(* CoDeSys 2.3.9.31 project: tcWiesenrain23.pro *)
(* Libraries: C:\Users\root\Desktop\nww.wiesenrain23\lib\oscat_building_100.lib 12.1.13 01:09:34, C:\Users\root\Desktop\nww.wiesenrain23\lib\oscat_basic_333.lib 12.1.13 01:05:45, C:\Users\root\Desktop\nww.wiesenrain23\lib\ModbusRTU.lib 29.12.13 03:10:52, STANDARD.LIB 5.6.98 11:03:02, TcBase.lib 14.5.09 11:14:08, TcEtherCAT.lib 8.3.12 16:06:42, TcSUPS.lib 22.3.10 12:59:22, TcSystem.lib 27.2.12 14:08:36, TcUtilities.lib 10.1.13 19:12:12 *)

(* Task configuration *)
TASK Standard (PRIORITY := 1, INTERVAL := T#10ms);
	MAIN
END_TASK
TASK Slow (PRIORITY := 2, INTERVAL := T#200ms);
	MAIN_SLOW
END_TASK
TASK Fast (PRIORITY := 0, INTERVAL := T#1ms);
	MAIN_FAST
END_TASK

(* Global variable list: Global_Variables *)
VAR_GLOBAL
	A_TemperatureUnit: ARRAY [0..7] OF ST_TemperatureUnit := (
			id := KELVIN,   (* commonly used in scientific endeavors *)
			unit := 'Kelvin',
			symbol := 'K',
			f1 := 0,
			f2 := 273.16,
			offset := 0,
			scale := 1,
			inventor := 'William Thomson, 1st Baron Kelvin'
		), (
			id := GRAD_CELSIUS,   (* used by most of the world's population *)
			unit := 'Celsius',
			symbol := '°C',
			f1 := 0,
			f2 := 100,
			offset := 273.15,
			scale := 1,
			inventor := 'Anders Celsius'
		), (
			id := GRAD_FAHRENHEIT,   (* commonly used in the United States *)
			unit := 'Fahrenheit',
			symbol := '°F',
			f1 := 0,
			f2 := 96,
			offset := 255.3722222222222, (* 459.67 * 5 / 9 *)
			scale := 0.55555555555555555555,
			inventor := 'Daniel Gabriel Fahrenheit'
		), (
			id := GRAD_RANKINE,
			unit := 'Rankine',
			symbol := '°Ra',
			f1 := 0,
			f2 := 96,
			offset := 0,
			scale := 0.5555555555555555555,
			inventor := 'William John Macquorn Rankine'
		), (
			id := GRAD_DELISLE,
			unit := 'Delisle',
			symbol := '°De',
			f1 := 150,
			f2 := 0,
			offset := 373.15,
			scale := -0.66666666666666666666,
			inventor := 'Joseph-Nicolas Delisle'
		), (
			id := GRAD_REAUMUR,
			unit := 'Réaumur',
			symbol := '°Ré',
			f1 := 0,
			f2 := 80,
			offset := 273.15,
			scale := 1.25,
			inventor := 'René-Antoine Ferchault de Réaumur'
		), (
			id := GRAD_NEWTON,
			unit := 'Newton',
			symbol := '°N',
			f1 := 0,
			f2 := 33,
			offset := 273.15,
			scale := 0.66666666666666666666,
			inventor := 'Sir Isaac Newton'
		), (
			id := GRAD_ROMER,
			unit := 'Rømer',
			symbol := '°Rø',
			f1 := 0,
			f2 := 60,
			offset := 258.86428571428571428572, (* 273.15 - 7.5 * 40 / 21 *)
			scale := 1.90476190476190476190,
			inventor := 'Ole Christensen Rømer'
		);
END_VAR

(* Global variable list: Global_Variables_MODBUS *)
VAR_GLOBAL CONSTANT
	uiMaxCurrentDeviceSpace: UDINT := 99;
END_VAR

(* Global variable list: TwinCAT_Configuration *)
(* Generated automatically by TwinCAT - (read only) *)
VAR_CONFIG
	MAIN._bwmAussenW AT %IX296.0 : BOOL;
	MAIN._bwmAussenSO AT %IX296.1 : BOOL;
	MAIN._bwmEgGang AT %IX124.0 : BOOL;	(*  ~ {LinkedWith:TIID^KG-HV A1 X001 EtherCAT [rechts]^OG-UV A1 Ethercat->K-Bus [unten links] ^OG-UV A7^Kanal 9^EG-Gang BWM} *)
	MAIN._bwmEgWc AT %IX128.0 : BOOL;	(*  ~ {LinkedWith:TIID^KG-HV A1 X001 EtherCAT [rechts]^OG-UV A1 Ethercat->K-Bus [unten links] ^OG-UV A7^Kanal 11^EG-WC BWM} *)
	MAIN._bwmHobby AT %IX108.0 : BOOL;	(*  ~ {LinkedWith:TIID^KG-HV A1 X001 EtherCAT [rechts]^KG-HV A35 EtherCat->E-Bus [links]^KG-HV A? E-Bus->K-Bus^KG-HV A5^Kanal 1^Hobby BWM} *)
	MAIN._bwmKgGang AT %IX76.0 : BOOL;	(*  ~ {LinkedWith:TIID^KG-HV A1 K-Bus [rechts]^KG-HV A1 (K-Bus)^KG-HV A33^Kanal 2^KG-Gang BWM} *)
	MAIN._bwmKochen AT %IX206.0 : BOOL;	(*  ~ {LinkedWith:TIID^KG-HV A1 X001 EtherCAT [rechts]^OG-UV A1 Ethercat->K-Bus [unten links] ^OG-UV A7^Kanal 10^Kochen BWM} *)
	MAIN._bwmLager AT %IX108.1 : BOOL;	(*  ~ {LinkedWith:TIID^KG-HV A1 X001 EtherCAT [rechts]^KG-HV A35 EtherCat->E-Bus [links]^KG-HV A? E-Bus->K-Bus^KG-HV A5^Kanal 5^Lager BWM} *)
	MAIN._bwmOgGang AT %IX120.0 : BOOL;	(*  ~ {LinkedWith:TIID^KG-HV A1 X001 EtherCAT [rechts]^OG-UV A1 Ethercat->K-Bus [unten links] ^OG-UV A7^Kanal 16^OG-Gang BWM} *)
	MAIN._bwmWaschen AT %IX112.0 : BOOL;	(*  ~ {LinkedWith:TIID^KG-HV A1 X001 EtherCAT [rechts]^KG-HV A35 EtherCat->E-Bus [links]^KG-HV A? E-Bus->K-Bus^KG-HV A5^Kanal 2^Waschen BWM} *)
	MAIN._lichtEgGang_status AT %IB300 : USINT;	(*  ~ {LinkedWith:TIID^KG-HV A1 X001 EtherCAT [rechts]^OG-UV A? Ethercat->K-Bus [mitte rechts]^OG-UV A9a^Kanal 2^EgGang Licht Status} *)
	MAIN._lichtEgGang_dataIn AT %IB301 : INT;	(*  ~ {LinkedWith:TIID^KG-HV A1 X001 EtherCAT [rechts]^OG-UV A? Ethercat->K-Bus [mitte rechts]^OG-UV A9a^Kanal 2^EgGang Licht DataIn} *)
	MAIN._lichtEgWc_status AT %IB303 : USINT;	(*  ~ {LinkedWith:TIID^KG-HV A1 X001 EtherCAT [rechts]^OG-UV A? Ethercat->K-Bus [mitte rechts]^OG-UV A9b^Kanal 2^EgWc Licht Status} *)
	MAIN._lichtEgWc_dataIn AT %IB304 : INT;	(*  ~ {LinkedWith:TIID^KG-HV A1 X001 EtherCAT [rechts]^OG-UV A? Ethercat->K-Bus [mitte rechts]^OG-UV A9b^Kanal 2^EgWc Licht Daten Ein} *)
	MAIN._lichtHobby_status AT %IB306 : USINT;
	MAIN._lichtHobby_dataIn AT %IB307 : INT;
	MAIN._lichtKochen_status AT %IB309 : USINT;
	MAIN._lichtKochen_dataIn AT %IB310 : INT;
	MAIN._lichtLager_status AT %IB312 : USINT;
	MAIN._lichtLager_dataIn AT %IB313 : INT;
	MAIN._lichtOgGang_status AT %IB315 : USINT;
	MAIN._lichtOgGang_dataIn AT %IB316 : INT;
	MAIN._lichtWaschen_status AT %IB318 : USINT;	(*  ~ {LinkedWith:TIID^KG-HV A1 X001 EtherCAT [rechts]^KG-HV A35 EtherCat->E-Bus [links]^KG-HV A? E-Bus->K-Bus^KG-HV A8b^Kanal 2^Waschen Licht Status} *)
	MAIN._lichtWaschen_dataIn AT %IB319 : INT;	(*  ~ {LinkedWith:TIID^KG-HV A1 X001 EtherCAT [rechts]^KG-HV A35 EtherCat->E-Bus [links]^KG-HV A? E-Bus->K-Bus^KG-HV A8b^Kanal 2^Waschen Licht Daten Ein} *)
	MAIN._temperaturArbeiten_status AT %IB324 : USINT;	(*  ~ {LinkedWith:TIID^KG-HV A1 X001 EtherCAT [rechts]^OG-UV A? Ethercat->K-Bus [mitte rechts]^OG-UV A74a^Kanal 2^Arbeiten Temperatur Status} *)
	MAIN._temperaturArbeiten_dataIn AT %IB325 : INT;	(*  ~ {LinkedWith:TIID^KG-HV A1 X001 EtherCAT [rechts]^OG-UV A? Ethercat->K-Bus [mitte rechts]^OG-UV A74a^Kanal 2^Arbeiten Temperatur Daten Ein} *)
	MAIN._temperaturEgBad_status AT %IB327 : USINT;
	MAIN._temperaturEgBad_dataIn AT %IB328 : INT;
	MAIN._temperaturEgGangSM_status AT %IB330 : USINT;	(*  ~ {LinkedWith:TIID^KG-HV A1 X001 EtherCAT [rechts]^OG-UV A? Ethercat->K-Bus [mitte rechts]^OG-UV A9a^Kanal 1^EgGang TemperaturSM Status} *)
	MAIN._temperaturEgGangSM_dataIn AT %IB331 : INT;	(*  ~ {LinkedWith:TIID^KG-HV A1 X001 EtherCAT [rechts]^OG-UV A? Ethercat->K-Bus [mitte rechts]^OG-UV A9a^Kanal 1^EgGang TemperaturSM DataIn} *)
	MAIN._temperaturEgGangSO_status AT %IB333 : USINT;
	MAIN._temperaturEgGangSO_dataIn AT %IB334 : INT;
	MAIN._temperaturEgWc_status AT %IB336 : USINT;	(*  ~ {LinkedWith:TIID^KG-HV A1 X001 EtherCAT [rechts]^OG-UV A? Ethercat->K-Bus [mitte rechts]^OG-UV A9b^Kanal 1^EgWc Temperatur Status} *)
	MAIN._temperaturEgWc_dataIn AT %IB337 : INT;	(*  ~ {LinkedWith:TIID^KG-HV A1 X001 EtherCAT [rechts]^OG-UV A? Ethercat->K-Bus [mitte rechts]^OG-UV A9b^Kanal 1^EgWc Temperatur Daten Ein} *)
	MAIN._temperaturEssen_status AT %IB339 : USINT;
	MAIN._temperaturEssen_dataIn AT %IB340 : INT;
	MAIN._temperaturGaeste_status AT %IB342 : USINT;
	MAIN._temperaturGaeste_dataIn AT %IB343 : INT;
	MAIN._temperaturHobby_status AT %IB345 : USINT;
	MAIN._temperaturHobby_dataIn AT %IB346 : INT;
	MAIN._temperaturKochen_status AT %IB348 : USINT;
	MAIN._temperaturKochen_dataIn AT %IB349 : INT;
	MAIN._temperaturLager_status AT %IB351 : USINT;
	MAIN._temperaturLager_dataIn AT %IB352 : INT;
	MAIN._temperaturOgBad_status AT %IB354 : USINT;
	MAIN._temperaturOgBad_dataIn AT %IB355 : INT;
	MAIN._temperaturOgGang_status AT %IB357 : USINT;	(*  ~ {LinkedWith:TIID^KG-HV A1 X001 EtherCAT [rechts]^OG-UV A? Ethercat->K-Bus [mitte rechts]^OG-UV A73a^Kanal 1^OgGang Temperatur Status} *)
	MAIN._temperaturOgGang_dataIn AT %IB358 : INT;	(*  ~ {LinkedWith:TIID^KG-HV A1 X001 EtherCAT [rechts]^OG-UV A? Ethercat->K-Bus [mitte rechts]^OG-UV A73a^Kanal 1^OgGang Temperatur Daten Ein} *)
	MAIN._temperaturOgKind_status AT %IB360 : USINT;
	MAIN._temperaturOgKind_dataIn AT %IB361 : INT;
	MAIN._temperaturOgWc_status AT %IB363 : USINT;
	MAIN._temperaturOgWc_dataIn AT %IB364 : INT;
	MAIN._temperaturSchlafen_status AT %IB366 : USINT;	(*  ~ {LinkedWith:TIID^KG-HV A1 X001 EtherCAT [rechts]^OG-UV A? Ethercat->K-Bus [mitte rechts]^OG-UV A10a^Kanal 1^Schlafen Temperatur Status} *)
	MAIN._temperaturSchlafen_dataIn AT %IB367 : INT;	(*  ~ {LinkedWith:TIID^KG-HV A1 X001 EtherCAT [rechts]^OG-UV A? Ethercat->K-Bus [mitte rechts]^OG-UV A10a^Kanal 1^Schlafen Temperatur DataIn} *)
	MAIN._temperaturVorrat_status AT %IB369 : USINT;
	MAIN._temperaturVorrat_dataIn AT %IB370 : INT;
	MAIN._temperaturWaschenON_status AT %IB372 : USINT;	(*  ~ {LinkedWith:TIID^KG-HV A1 X001 EtherCAT [rechts]^KG-HV A35 EtherCat->E-Bus [links]^KG-HV A? E-Bus->K-Bus^KG-HV A8b^Kanal 1^WaschenO TemperaturN Status} *)
	MAIN._temperaturWaschenON_dataIn AT %IB373 : INT;	(*  ~ {LinkedWith:TIID^KG-HV A1 X001 EtherCAT [rechts]^KG-HV A35 EtherCat->E-Bus [links]^KG-HV A? E-Bus->K-Bus^KG-HV A8b^Kanal 1^WaschenO TemperaturN Daten Ein} *)
	MAIN._temperaturWaschenOS_status AT %IB375 : USINT;
	MAIN._temperaturWaschenOS_dataIn AT %IB376 : INT;
	MAIN._temperaturWohnen_status AT %IB378 : USINT;	(*  ~ {LinkedWith:TIID^KG-HV A1 X001 EtherCAT [rechts]^OG-UV A? Ethercat->K-Bus [mitte rechts]^OG-UV A10a^Kanal 2^Wohnen Temperatur Status} *)
	MAIN._temperaturWohnen_dataIn AT %IB379 : INT;	(*  ~ {LinkedWith:TIID^KG-HV A1 X001 EtherCAT [rechts]^OG-UV A? Ethercat->K-Bus [mitte rechts]^OG-UV A10a^Kanal 2^Wohnen Temperatur DataIn} *)
	MAIN._tasterArbeitenOO AT %IX206.1 : BOOL;	(*  ~ {LinkedWith:TIID^KG-HV A1 X001 EtherCAT [rechts]^OG-UV A1 Ethercat->K-Bus [unten links] ^OG-UV A6^Kanal 3^ArbeitenO TasterO} *)
	MAIN._tasterArbeitenOL AT %IX206.2 : BOOL;	(*  ~ {LinkedWith:TIID^KG-HV A1 X001 EtherCAT [rechts]^OG-UV A1 Ethercat->K-Bus [unten links] ^OG-UV A6^Kanal 4^ArbeitenO TasterL} *)
	MAIN._tasterArbeitenOR AT %IX206.3 : BOOL;	(*  ~ {LinkedWith:TIID^KG-HV A1 X001 EtherCAT [rechts]^OG-UV A1 Ethercat->K-Bus [unten links] ^OG-UV A6^Kanal 5^ArbeitenO TasterR} *)
	MAIN._tasterArbeitenSL AT %IX206.4 : BOOL;	(*  ~ {LinkedWith:TIID^KG-HV A1 X001 EtherCAT [rechts]^OG-UV A1 Ethercat->K-Bus [unten links] ^OG-UV A5^Kanal 11^ArbeitenS TasterL} *)
	MAIN._tasterArbeitenSR AT %IX206.5 : BOOL;	(*  ~ {LinkedWith:TIID^KG-HV A1 X001 EtherCAT [rechts]^OG-UV A1 Ethercat->K-Bus [unten links] ^OG-UV A5^Kanal 12^ArbeitenS TasterR} *)
	MAIN._tasterDgKind AT %IX206.6 : BOOL;
	MAIN._tasterEgBadL AT %IX132.1 : BOOL;	(*  ~ {LinkedWith:TIID^KG-HV A1 X001 EtherCAT [rechts]^OG-UV A1 Ethercat->K-Bus [unten links] ^OG-UV A5^Kanal 7^EG-Bad TasterL} *)
	MAIN._tasterEgBadR AT %IX132.0 : BOOL;	(*  ~ {LinkedWith:TIID^KG-HV A1 X001 EtherCAT [rechts]^OG-UV A1 Ethercat->K-Bus [unten links] ^OG-UV A5^Kanal 8^EG-Bad TasterR} *)
	MAIN._tasterEgGang AT %IX80.0 : BOOL;	(*  ~ {LinkedWith:TIID^KG-HV A1 K-Bus [rechts]^KG-HV A1 (K-Bus)^KG-HV A4^Kanal 10^EG-Gang Taster} *)
	MAIN._tasterEgWc AT %IX128.1 : BOOL;	(*  ~ {LinkedWith:TIID^KG-HV A1 X001 EtherCAT [rechts]^OG-UV A1 Ethercat->K-Bus [unten links] ^OG-UV A5^Kanal 6^EG-WC Taster} *)
	MAIN._tasterEssenO AT %IX140.0 : BOOL;	(*  ~ {LinkedWith:TIID^KG-HV A1 X001 EtherCAT [rechts]^OG-UV A1 Ethercat->K-Bus [unten links] ^OG-UV A4^Kanal 6^EssenS TasterO} *)
	MAIN._tasterEssenL AT %IX140.1 : BOOL;	(*  ~ {LinkedWith:TIID^KG-HV A1 X001 EtherCAT [rechts]^OG-UV A1 Ethercat->K-Bus [unten links] ^OG-UV A4^Kanal 7^EssenS TasterL} *)
	MAIN._tasterEssenR AT %IX140.2 : BOOL;	(*  ~ {LinkedWith:TIID^KG-HV A1 X001 EtherCAT [rechts]^OG-UV A1 Ethercat->K-Bus [unten links] ^OG-UV A4^Kanal 8^EssenS TasterR} *)
	MAIN._tasterGaesteO AT %IX136.0 : BOOL;	(*  ~ {LinkedWith:TIID^KG-HV A1 K-Bus [rechts]^KG-HV A1 (K-Bus)^OG-UV A72^Kanal 1^GaesteN TasterO} *)
	MAIN._tasterGaesteL AT %IX136.1 : BOOL;	(*  ~ {LinkedWith:TIID^KG-HV A1 K-Bus [rechts]^KG-HV A1 (K-Bus)^OG-UV A72^Kanal 2^GaesteN TasterL} *)
	MAIN._tasterGaesteR AT %IX136.2 : BOOL;	(*  ~ {LinkedWith:TIID^KG-HV A1 K-Bus [rechts]^KG-HV A1 (K-Bus)^OG-UV A72^Kanal 3^GaesteN TasterR} *)
	MAIN._tasterHeizen AT %IX76.1 : BOOL;	(*  ~ {LinkedWith:TIID^KG-HV A1 K-Bus [rechts]^KG-HV A1 (K-Bus)^KG-HV A4^Kanal 7^Heizen Taster} *)
	MAIN._tasterHobbyL AT %IX76.2 : BOOL;	(*  ~ {LinkedWith:TIID^KG-HV A1 K-Bus [rechts]^KG-HV A1 (K-Bus)^KG-HV A4^Kanal 5^Hobby TasterL} *)
	MAIN._tasterHobbyR AT %IX76.3 : BOOL;	(*  ~ {LinkedWith:TIID^KG-HV A1 K-Bus [rechts]^KG-HV A1 (K-Bus)^KG-HV A4^Kanal 6^Hobby TasterR} *)
	MAIN._tasterKochenOL AT %IX144.0 : BOOL;	(*  ~ {LinkedWith:TIID^KG-HV A1 X001 EtherCAT [rechts]^OG-UV A1 Ethercat->K-Bus [unten links] ^OG-UV A4^Kanal 4^KochenO TasterL} *)
	MAIN._tasterKochenOR AT %IX144.1 : BOOL;	(*  ~ {LinkedWith:TIID^KG-HV A1 X001 EtherCAT [rechts]^OG-UV A1 Ethercat->K-Bus [unten links] ^OG-UV A4^Kanal 5^KochenO TasterR} *)
	MAIN._tasterKochenWO AT %IX144.2 : BOOL;	(*  ~ {LinkedWith:TIID^KG-HV A1 X001 EtherCAT [rechts]^OG-UV A1 Ethercat->K-Bus [unten links] ^OG-UV A4^Kanal 1^KochenW TasterO} *)
	MAIN._tasterKochenWL AT %IX144.3 : BOOL;	(*  ~ {LinkedWith:TIID^KG-HV A1 X001 EtherCAT [rechts]^OG-UV A1 Ethercat->K-Bus [unten links] ^OG-UV A4^Kanal 2^KochenW TasterL} *)
	MAIN._tasterKochenWR AT %IX144.4 : BOOL;	(*  ~ {LinkedWith:TIID^KG-HV A1 X001 EtherCAT [rechts]^OG-UV A1 Ethercat->K-Bus [unten links] ^OG-UV A4^Kanal 3^KochenW TasterR} *)
	MAIN._tasterLagerNO AT %IX76.6 : BOOL;	(*  ~ {LinkedWith:TIID^KG-HV A1 K-Bus [rechts]^KG-HV A1 (K-Bus)^KG-HV A4^Kanal 9^LagerNO Taster} *)
	MAIN._tasterLagerS AT %IX76.7 : BOOL;	(*  ~ {LinkedWith:TIID^KG-HV A1 K-Bus [rechts]^KG-HV A1 (K-Bus)^KG-HV A4^Kanal 8^LagerS Taster} *)
	MAIN._tasterOgBadL AT %IX206.7 : BOOL;
	MAIN._tasterOgBadR AT %IX207.0 : BOOL;
	MAIN._tasterOgKindNO AT %IX207.1 : BOOL;
	MAIN._tasterOgKindNL AT %IX207.2 : BOOL;
	MAIN._tasterOgKindNR AT %IX207.3 : BOOL;
	MAIN._tasterOgKindWL AT %IX207.4 : BOOL;	(*  ~ {LinkedWith:TIID^KG-HV A1 X001 EtherCAT [rechts]^OG-UV A1 Ethercat->K-Bus [unten links] ^OG-UV A5^Kanal 9^OG-KindW TasterL} *)
	MAIN._tasterOgKindWR AT %IX207.5 : BOOL;	(*  ~ {LinkedWith:TIID^KG-HV A1 X001 EtherCAT [rechts]^OG-UV A1 Ethercat->K-Bus [unten links] ^OG-UV A5^Kanal 10^OG-KindW TasteR} *)
	MAIN._tasterOgWc AT %IX207.6 : BOOL;
	MAIN._tasterSchlafenOo AT %IX408.0 : BOOL;	(*  ~ {LinkedWith:TIID^KG-HV A1 X001 EtherCAT [rechts]^OG-UV A1 Ethercat->K-Bus [unten links] ^OG-UV A4^Kanal 12^SchlafenO TasterO} *)
	MAIN._tasterSchlafenOl AT %IX408.1 : BOOL;	(*  ~ {LinkedWith:TIID^KG-HV A1 X001 EtherCAT [rechts]^OG-UV A1 Ethercat->K-Bus [unten links] ^OG-UV A4^Kanal 13^SchlafenO TasterL} *)
	MAIN._tasterSchlafenOr AT %IX408.2 : BOOL;	(*  ~ {LinkedWith:TIID^KG-HV A1 X001 EtherCAT [rechts]^OG-UV A1 Ethercat->K-Bus [unten links] ^OG-UV A4^Kanal 14^SchlafenO TasterR} *)
	MAIN._tasterSchlafenWML AT %IX116.3 : BOOL;	(*  ~ {LinkedWith:TIID^KG-HV A1 X001 EtherCAT [rechts]^OG-UV A1 Ethercat->K-Bus [unten links] ^OG-UV A4^Kanal 15^SchlafenWM TasterL} *)
	MAIN._tasterSchlafenWMR AT %IX116.4 : BOOL;	(*  ~ {LinkedWith:TIID^KG-HV A1 X001 EtherCAT [rechts]^OG-UV A1 Ethercat->K-Bus [unten links] ^OG-UV A4^Kanal 16^SchlafenWM TasterR} *)
	MAIN._tasterSchlafenWNL AT %IX116.5 : BOOL;	(*  ~ {LinkedWith:TIID^KG-HV A1 X001 EtherCAT [rechts]^OG-UV A1 Ethercat->K-Bus [unten links] ^OG-UV A5^Kanal 1^SchlafenWN TasterL} *)
	MAIN._tasterSchlafenWNR AT %IX116.6 : BOOL;	(*  ~ {LinkedWith:TIID^KG-HV A1 X001 EtherCAT [rechts]^OG-UV A1 Ethercat->K-Bus [unten links] ^OG-UV A5^Kanal 2^SchlafenWN TasterR} *)
	MAIN._tasterSpeis AT %IX207.7 : BOOL;	(*  ~ {LinkedWith:TIID^KG-HV A1 X001 EtherCAT [rechts]^OG-UV A1 Ethercat->K-Bus [unten links] ^OG-UV A5^Kanal 16^Speis Tuerkontakt} *)
	MAIN._tasterWaschenL AT %IX76.4 : BOOL;	(*  ~ {LinkedWith:TIID^KG-HV A1 K-Bus [rechts]^KG-HV A1 (K-Bus)^KG-HV A4^Kanal 3^Waschen TasterL} *)
	MAIN._tasterWaschenR AT %IX76.5 : BOOL;	(*  ~ {LinkedWith:TIID^KG-HV A1 K-Bus [rechts]^KG-HV A1 (K-Bus)^KG-HV A4^Kanal 4^Waschen TasterR} *)
	MAIN._tasterWohnenOO AT %IX124.1 : BOOL;	(*  ~ {LinkedWith:TIID^KG-HV A1 X001 EtherCAT [rechts]^OG-UV A1 Ethercat->K-Bus [unten links] ^OG-UV A4^Kanal 9^WohnenO TasterO} *)
	MAIN._tasterWohnenOL AT %IX124.2 : BOOL;	(*  ~ {LinkedWith:TIID^KG-HV A1 X001 EtherCAT [rechts]^OG-UV A1 Ethercat->K-Bus [unten links] ^OG-UV A4^Kanal 10^WohnenO TasterL} *)
	MAIN._tasterWohnenOR AT %IX124.3 : BOOL;	(*  ~ {LinkedWith:TIID^KG-HV A1 X001 EtherCAT [rechts]^OG-UV A1 Ethercat->K-Bus [unten links] ^OG-UV A4^Kanal 11^WohnenO TasterR} *)
	MAIN._tasterWohnenWO AT %IX124.4 : BOOL;	(*  ~ {LinkedWith:TIID^KG-HV A1 X001 EtherCAT [rechts]^OG-UV A1 Ethercat->K-Bus [unten links] ^OG-UV A5^Kanal 3^WohnenW TasterO} *)
	MAIN._tasterWohnenWL AT %IX124.5 : BOOL;	(*  ~ {LinkedWith:TIID^KG-HV A1 X001 EtherCAT [rechts]^OG-UV A1 Ethercat->K-Bus [unten links] ^OG-UV A5^Kanal 4^WohnenW TasterL} *)
	MAIN._tasterWohnenWR AT %IX124.6 : BOOL;	(*  ~ {LinkedWith:TIID^KG-HV A1 X001 EtherCAT [rechts]^OG-UV A1 Ethercat->K-Bus [unten links] ^OG-UV A5^Kanal 5^WohnenW TasterR} *)
	MAIN._dimmerWohnenN_intensity AT %IB208 : REAL;
	MAIN._dimmerWohnenN_status AT %IB212 : USINT;	(*  ~ {LinkedWith:TIID^KG-HV A1 X001 EtherCAT [rechts]^OG-UV A? Ethercat->K-Bus [mitte rechts]^OG-UV A29^Kanal 1^WohnenM Lampe Status} *)
	MAIN._dimmerWohnenN_dataIn AT %IB213 : INT;	(*  ~ {LinkedWith:TIID^KG-HV A1 X001 EtherCAT [rechts]^OG-UV A? Ethercat->K-Bus [mitte rechts]^OG-UV A29^Kanal 1^WohnenM Lampe DataIn} *)
	MAIN._dimmerWohnenN_dataOut AT %QB24 : INT;	(*  ~ {LinkedWith:TIID^KG-HV A1 X001 EtherCAT [rechts]^OG-UV A? Ethercat->K-Bus [mitte rechts]^OG-UV A29^Kanal 1^WohnenM Lampe DataOut} *)
	MAIN._dimmerWohnenN_control AT %QB26 : USINT;	(*  ~ {LinkedWith:TIID^KG-HV A1 X001 EtherCAT [rechts]^OG-UV A? Ethercat->K-Bus [mitte rechts]^OG-UV A29^Kanal 1^WohnenM Lampe Control} *)
	MAIN._dimmerEgBadSM_intensity AT %IB216 : REAL;
	MAIN._dimmerEgBadSM_status AT %IB220 : USINT;	(*  ~ {LinkedWith:TIID^KG-HV A1 X001 EtherCAT [rechts]^OG-UV A? Ethercat->K-Bus [mitte rechts]^OG-UV A32^Kanal 1^EgBad LichtSM Status} *)
	MAIN._dimmerEgBadSM_dataIn AT %IB221 : INT;	(*  ~ {LinkedWith:TIID^KG-HV A1 X001 EtherCAT [rechts]^OG-UV A? Ethercat->K-Bus [mitte rechts]^OG-UV A32^Kanal 1^EgBad LichtSM Daten Ein} *)
	MAIN._dimmerEgBadSM_dataOut AT %QB36 : INT;	(*  ~ {LinkedWith:TIID^KG-HV A1 X001 EtherCAT [rechts]^OG-UV A? Ethercat->K-Bus [mitte rechts]^OG-UV A32^Kanal 1^EgBad LichtSM Daten Aus} *)
	MAIN._dimmerEgBadSM_control AT %QB38 : USINT;	(*  ~ {LinkedWith:TIID^KG-HV A1 X001 EtherCAT [rechts]^OG-UV A? Ethercat->K-Bus [mitte rechts]^OG-UV A32^Kanal 1^EgBad LichtSM Kontrolle} *)
	MAIN._lampeEgBadOM AT %QX20.1 : BOOL;	(*  ~ {LinkedWith:TIID^KG-HV A1 X001 EtherCAT [rechts]^OG-UV A1 Ethercat->K-Bus [unten links] ^OG-UV A31^Kanal 2^EG-BadOM Lampe} *)
	MAIN._lampeEgGang AT %QX20.2 : BOOL;	(*  ~ {LinkedWith:TIID^KG-HV A1 X001 EtherCAT [rechts]^OG-UV A1 Ethercat->K-Bus [unten links] ^OG-UV A24^Kanal 1^EG-Gang Lampen} *)
	MAIN._lampeEgWc AT %QX20.3 : BOOL;	(*  ~ {LinkedWith:TIID^KG-HV A1 X001 EtherCAT [rechts]^OG-UV A1 Ethercat->K-Bus [unten links] ^OG-UV A31^Kanal 1^EG-WC Lampe} *)
	MAIN._lampeEssenM AT %QX20.4 : BOOL;	(*  ~ {LinkedWith:TIID^KG-HV A1 X001 EtherCAT [rechts]^OG-UV A1 Ethercat->K-Bus [unten links] ^OG-UV A14^Kanal 1^EssenM Lampe} *)
	MAIN._lampeEssenS AT %QX20.5 : BOOL;	(*  ~ {LinkedWith:TIID^KG-HV A1 X001 EtherCAT [rechts]^OG-UV A1 Ethercat->K-Bus [unten links] ^OG-UV A14^Kanal 2^EssenS Lampe} *)
	MAIN._lampeKochenSW AT %QX32.0 : BOOL;	(*  ~ {LinkedWith:TIID^KG-HV A1 X001 EtherCAT [rechts]^OG-UV A1 Ethercat->K-Bus [unten links] ^OG-UV A24^Kanal 2^KochenSW Lampe} *)
	MAIN._lampeOgGang AT %QX20.6 : BOOL;	(*  ~ {LinkedWith:TIID^KG-HV A1 K-Bus [rechts]^KG-HV A1 (K-Bus)^OG-UV A40^Kanal 1^OG-Gang Lampe} *)
	MAIN._lampeEgOgStiege AT %QX52.0 : BOOL;	(*  ~ {LinkedWith:TIID^KG-HV A1 K-Bus [rechts]^KG-HV A1 (K-Bus)^OG-UV A40^Kanal 2^EG-OG-Stiege Lampe} *)
	MAIN._lampeSchlafenS AT %QX20.0 : BOOL;	(*  ~ {LinkedWith:TIID^KG-HV A1 X001 EtherCAT [rechts]^OG-UV A1 Ethercat->K-Bus [unten links] ^OG-UV A28^Kanal 1^SchlafenS Lampen} *)
	MAIN._lampeWohnenM AT %QX28.0 : BOOL;	(*  ~ {LinkedWith:TIID^KG-HV A1 X001 EtherCAT [rechts]^OG-UV A1 Ethercat->K-Bus [unten links] ^OG-UV A28^Kanal 2^WohnenM Lampe} *)
	MAIN.heizenHK1.mischer AT %QB12 : INT;
	MAIN.heizenHK1.pumpe AT %QB14 : INT;
	MAIN.heizenHK2.mischer AT %QB16 : INT;
	MAIN.heizenHK2.pumpe AT %QB18 : INT;
	MAIN.egBadJalousie.Qu AT %QX92.0 : BOOL;	(*  ~ {LinkedWith:TIID^KG-HV A1 K-Bus [rechts]^KG-HV A1 (K-Bus)^OG-UV A59^Kanal 1^EG-Bad JalousieAuf} *)
	MAIN.egBadJalousie.Qd AT %QX92.1 : BOOL;	(*  ~ {LinkedWith:TIID^KG-HV A1 K-Bus [rechts]^KG-HV A1 (K-Bus)^OG-UV A59^Kanal 2^EG-Bad JalousieAb} *)
	MAIN.essenJalousie.Qu AT %QX92.2 : BOOL;	(*  ~ {LinkedWith:TIID^KG-HV A1 X001 EtherCAT [rechts]^OG-UV A1 Ethercat->K-Bus [unten links] ^OG-UV A65^Kanal 1^Essen JalousieAuf} *)
	MAIN.essenJalousie.Qd AT %QX92.3 : BOOL;	(*  ~ {LinkedWith:TIID^KG-HV A1 X001 EtherCAT [rechts]^OG-UV A1 Ethercat->K-Bus [unten links] ^OG-UV A65^Kanal 2^Essen JalousieAb} *)
	MAIN.kochenJalousieS.Qu AT %QX92.4 : BOOL;	(*  ~ {LinkedWith:TIID^KG-HV A1 X001 EtherCAT [rechts]^OG-UV A1 Ethercat->K-Bus [unten links] ^OG-UV A66^Kanal 1^KochenS JalousieAuf} *)
	MAIN.kochenJalousieS.Qd AT %QX92.5 : BOOL;	(*  ~ {LinkedWith:TIID^KG-HV A1 X001 EtherCAT [rechts]^OG-UV A1 Ethercat->K-Bus [unten links] ^OG-UV A66^Kanal 2^KochenS JalousieAb} *)
	MAIN.kochenJalousieO.Qu AT %QX92.6 : BOOL;	(*  ~ {LinkedWith:TIID^KG-HV A1 X001 EtherCAT [rechts]^OG-UV A1 Ethercat->K-Bus [unten links] ^OG-UV A67^Kanal 1^KochenO JalousieAuf} *)
	MAIN.kochenJalousieO.Qd AT %QX92.7 : BOOL;	(*  ~ {LinkedWith:TIID^KG-HV A1 X001 EtherCAT [rechts]^OG-UV A1 Ethercat->K-Bus [unten links] ^OG-UV A67^Kanal 2^KochenO JalousieAb} *)
	MAIN.schlafenJalousieN.Qu AT %QX88.2 : BOOL;	(*  ~ {LinkedWith:TIID^KG-HV A1 K-Bus [rechts]^KG-HV A1 (K-Bus)^OG-UV A60^Kanal 1^SchlafenN JalousieAuf} *)
	MAIN.schlafenJalousieN.Qd AT %QX88.3 : BOOL;	(*  ~ {LinkedWith:TIID^KG-HV A1 K-Bus [rechts]^KG-HV A1 (K-Bus)^OG-UV A60^Kanal 2^SchlafenN JalousieAb} *)
	MAIN.schlafenJalousieW.Qu AT %QX88.4 : BOOL;	(*  ~ {LinkedWith:TIID^KG-HV A1 K-Bus [rechts]^KG-HV A1 (K-Bus)^OG-UV A61^Kanal 1^SchlafenW JalousieAuf} *)
	MAIN.schlafenJalousieW.Qd AT %QX88.5 : BOOL;	(*  ~ {LinkedWith:TIID^KG-HV A1 K-Bus [rechts]^KG-HV A1 (K-Bus)^OG-UV A61^Kanal 2^SchlafenW JalousieAb} *)
	MAIN.wohnenJalousieS.Qu AT %QX93.0 : BOOL;	(*  ~ {LinkedWith:TIID^KG-HV A1 X001 EtherCAT [rechts]^OG-UV A1 Ethercat->K-Bus [unten links] ^OG-UV A64^Kanal 1^WohnenS JalousieAuf} *)
	MAIN.wohnenJalousieS.Qd AT %QX93.1 : BOOL;	(*  ~ {LinkedWith:TIID^KG-HV A1 X001 EtherCAT [rechts]^OG-UV A1 Ethercat->K-Bus [unten links] ^OG-UV A64^Kanal 2^WohnenS JalousieAb} *)
	MAIN.wohnenJalousieWa.Qu AT %QX93.2 : BOOL;	(*  ~ {LinkedWith:TIID^KG-HV A1 K-Bus [rechts]^KG-HV A1 (K-Bus)^OG-UV A62^Kanal 1^WohnenWa JalousieAuf} *)
	MAIN.wohnenJalousieWa.Qd AT %QX93.3 : BOOL;	(*  ~ {LinkedWith:TIID^KG-HV A1 K-Bus [rechts]^KG-HV A1 (K-Bus)^OG-UV A62^Kanal 2^WohnenWa JalousieAb} *)
	MAIN.wohnenJalousieWb.Qu AT %QX93.4 : BOOL;	(*  ~ {LinkedWith:TIID^KG-HV A1 K-Bus [rechts]^KG-HV A1 (K-Bus)^OG-UV A63^Kanal 1^WohnenWb JalousieAuf} *)
	MAIN.wohnenJalousieWb.Qd AT %QX93.5 : BOOL;	(*  ~ {LinkedWith:TIID^KG-HV A1 K-Bus [rechts]^KG-HV A1 (K-Bus)^OG-UV A63^Kanal 2^WohnenWb JalousieAb} *)
	MAIN.arbeitenJalousieN.Qu AT %QX100.0 : BOOL;
	MAIN.arbeitenJalousieN.Qd AT %QX100.1 : BOOL;
	MAIN.arbeitenJalousieW.Qu AT %QX100.2 : BOOL;
	MAIN.arbeitenJalousieW.Qd AT %QX100.3 : BOOL;
	MAIN.arbeitenJalousieS.Qu AT %QX100.4 : BOOL;
	MAIN.arbeitenJalousieS.Qd AT %QX100.5 : BOOL;
	MAIN.gaesteJalousieO.Qu AT %QX100.6 : BOOL;
	MAIN.gaesteJalousieO.Qd AT %QX100.7 : BOOL;
	MAIN.gaesteJalousieS.Qu AT %QX101.0 : BOOL;
	MAIN.gaesteJalousieS.Qd AT %QX101.1 : BOOL;
	MAIN.ogBadJalousie.Qu AT %QX96.0 : BOOL;	(*  ~ {LinkedWith:TIID^KG-HV A1 K-Bus [rechts]^KG-HV A1 (K-Bus)^OG-UV A82^Kanal 1^OG-Bad JalousieAuf} *)
	MAIN.ogBadJalousie.Qd AT %QX96.1 : BOOL;	(*  ~ {LinkedWith:TIID^KG-HV A1 K-Bus [rechts]^KG-HV A1 (K-Bus)^OG-UV A82^Kanal 2^OG-Bad JalousieAb} *)
	MAIN.ogKindJalousieS.Qu AT %QX101.2 : BOOL;
	MAIN.ogKindJalousieS.Qd AT %QX101.3 : BOOL;
	MAIN.ogKindJalousieW.Qu AT %QX101.4 : BOOL;
	MAIN.ogKindJalousieW.Qd AT %QX101.5 : BOOL;
	MAIN_FAST.fbFroeling.modbusMaster.InData AT %IB384 : MB_KL6inData22B;
	MAIN_FAST.fbFroeling.modbusMaster.OutData AT %QB56 : MB_KL6outData22B;
	MAIN_FAST.uiStateCX5000 AT %IB224 : UINT;	(*  ~ {LinkedWith:TIID^KG-HV A1 K-Bus [rechts]^KG-HV A1 (K-Bus)^Eingänge^State} *)
	MAIN_FAST.uiControlCX5000 AT %QB40 : UINT;	(*  ~ {LinkedWith:TIID^KG-HV A1 K-Bus [rechts]^KG-HV A1 (K-Bus)^Ausgänge^Ctrl} *)
	MAIN_FAST.iVoltagePhase1 AT %IB226 : ARRAY [0..9] OF INT;	(*  ~ {LinkedWith:TIID^KG-HV A1 X001 EtherCAT [rechts]^KG-HV A35 EtherCat->E-Bus [links]^KG-HV A18^L1 Voltage Samples^U1 SAMPLES} *)
	MAIN_FAST.iVoltagePhase2 AT %IB246 : ARRAY [0..9] OF INT;	(*  ~ {LinkedWith:TIID^KG-HV A1 X001 EtherCAT [rechts]^KG-HV A35 EtherCat->E-Bus [links]^KG-HV A18^L2 Voltage Samples^U2 SAMPLES} *)
	MAIN_FAST.iVoltagePhase3 AT %IB266 : ARRAY [0..9] OF INT;	(*  ~ {LinkedWith:TIID^KG-HV A1 X001 EtherCAT [rechts]^KG-HV A35 EtherCat->E-Bus [links]^KG-HV A18^L3 Voltage Samples^U3 SAMPLES} *)
	MAIN_FAST.uliStartTimeNextLatch AT %IB286 : ARRAY [0..1] OF UDINT;	(*  ~ {LinkedWith:TIID^KG-HV A1 X001 EtherCAT [rechts]^KG-HV A35 EtherCat->E-Bus [links]^KG-HV A18^AI Timestamp NextSync1Time^StartTimeNextLatch} *)
	MAIN_FAST.bWcState AT %IX294.0 : BOOL;	(*  ~ {LinkedWith:TIID^KG-HV A1 X001 EtherCAT [rechts]^KG-HV A35 EtherCat->E-Bus [links]^KG-HV A18^WcState^WcState} *)
	MAIN_FAST.fbA28CH1.bRelay AT %QX42.0 : BOOL;	(*  ~ {LinkedWith:TIID^KG-HV A1 K-Bus [rechts]^KG-HV A1 (K-Bus)^KG-HV A28^Kanal 1^Heizen PumpeSolar} *)
	MAIN_FAST.fbA28CH2.bRelay AT %QX42.1 : BOOL;	(*  ~ {LinkedWith:TIID^KG-HV A1 K-Bus [rechts]^KG-HV A1 (K-Bus)^KG-HV A28^Kanal 2^Heizen PumpeWarmwasser} *)
	MAIN_FAST.fbA29CH1.bRelay AT %QX42.2 : BOOL;	(*  ~ {LinkedWith:TIID^KG-HV A1 K-Bus [rechts]^KG-HV A1 (K-Bus)^KG-HV A29^Kanal 1^Heizen PumpePufferladung} *)
	MAIN_FAST.fbA29CH2.bRelay AT %QX42.3 : BOOL;	(*  ~ {LinkedWith:TIID^KG-HV A1 K-Bus [rechts]^KG-HV A1 (K-Bus)^KG-HV A29^Kanal 2^Heizen PumpeHeizkreis2} *)
	MAIN_FAST.fbA30CH1.bRelay AT %QX42.4 : BOOL;	(*  ~ {LinkedWith:TIID^KG-HV A1 K-Bus [rechts]^KG-HV A1 (K-Bus)^KG-HV A30^Kanal 1^Heizen MischerPuffer} *)
	MAIN_FAST.fbA30CH2.bRelay AT %QX42.5 : BOOL;	(*  ~ {LinkedWith:TIID^KG-HV A1 K-Bus [rechts]^KG-HV A1 (K-Bus)^KG-HV A30^Kanal 2^Heizen MischerSolar} *)
	MAIN_FAST.fbA31CH1.bRelay AT %QX42.6 : BOOL;	(*  ~ {LinkedWith:TIID^KG-HV A1 K-Bus [rechts]^KG-HV A1 (K-Bus)^KG-HV A31 (reserve)^Kanal 1^Ausgang} *)
	MAIN_FAST.fbA31CH2.bRelay AT %QX42.7 : BOOL;	(*  ~ {LinkedWith:TIID^KG-HV A1 K-Bus [rechts]^KG-HV A1 (K-Bus)^KG-HV A31 (reserve)^Kanal 2^Ausgang} *)
	MAIN_FAST.fbA32CH1.bRelay AT %QX43.0 : BOOL;	(*  ~ {LinkedWith:TIID^KG-HV A1 K-Bus [rechts]^KG-HV A1 (K-Bus)^KG-HV A32^Kanal 1^Waschen Tauchpumpe} *)
	MAIN_FAST.fbA32CH2.bRelay AT %QX43.1 : BOOL;	(*  ~ {LinkedWith:TIID^KG-HV A1 K-Bus [rechts]^KG-HV A1 (K-Bus)^KG-HV A32^Kanal 2^Ausgang} *)
	MAIN_FAST.fbA20CH1.bRelay AT %QX43.2 : BOOL;	(*  ~ {LinkedWith:TIID^KG-HV A1 K-Bus [rechts]^KG-HV A1 (K-Bus)^KG-HV A20^Kanal 1^KG-Gang Lampe} *)
	MAIN_FAST.fbA20CH2.bRelay AT %QX43.3 : BOOL;	(*  ~ {LinkedWith:TIID^KG-HV A1 K-Bus [rechts]^KG-HV A1 (K-Bus)^KG-HV A20^Kanal 2^KG-EG-Stiege Lampe} *)
	MAIN_FAST.fbA21CH1.bRelay AT %QX43.4 : BOOL;	(*  ~ {LinkedWith:TIID^KG-HV A1 K-Bus [rechts]^KG-HV A1 (K-Bus)^KG-HV A21^Kanal 1^Lager Lampe} *)
	MAIN_FAST.fbA21CH2.bRelay AT %QX43.5 : BOOL;	(*  ~ {LinkedWith:TIID^KG-HV A1 K-Bus [rechts]^KG-HV A1 (K-Bus)^KG-HV A21^Kanal 2^Ausgang} *)
	MAIN_FAST.fbA23CH1.bRelay AT %QX43.6 : BOOL;	(*  ~ {LinkedWith:TIID^KG-HV A1 K-Bus [rechts]^KG-HV A1 (K-Bus)^KG-HV A23^Kanal 1^Heizen Lampe} *)
	MAIN_FAST.fbA23CH2.bRelay AT %QX43.7 : BOOL;	(*  ~ {LinkedWith:TIID^KG-HV A1 K-Bus [rechts]^KG-HV A1 (K-Bus)^KG-HV A23^Kanal 2^WaschenS Lampe} *)
	MAIN_FAST.fbA24CH1.bRelay AT %QX44.0 : BOOL;	(*  ~ {LinkedWith:TIID^KG-HV A1 K-Bus [rechts]^KG-HV A1 (K-Bus)^KG-HV A24^Kanal 1^WaschenN Lampe} *)
	MAIN_FAST.fbA24CH2.bRelay AT %QX44.1 : BOOL;	(*  ~ {LinkedWith:TIID^KG-HV A1 K-Bus [rechts]^KG-HV A1 (K-Bus)^KG-HV A24^Kanal 2^HobbyN Lampe} *)
	MAIN_FAST.fbA25CH1.bRelay AT %QX44.2 : BOOL;	(*  ~ {LinkedWith:TIID^KG-HV A1 K-Bus [rechts]^KG-HV A1 (K-Bus)^KG-HV A25^Kanal 1^Vorrat Lampe} *)
	MAIN_FAST.fbA25CH2.bRelay AT %QX44.3 : BOOL;	(*  ~ {LinkedWith:TIID^KG-HV A1 K-Bus [rechts]^KG-HV A1 (K-Bus)^KG-HV A25^Kanal 2^HobbyS Lampe} *)
	MAIN_FAST.fbA26CH1.bRelay AT %QX44.4 : BOOL;	(*  ~ {LinkedWith:TIID^KG-HV A1 K-Bus [rechts]^KG-HV A1 (K-Bus)^KG-HV A26^Kanal 1^Ausgang} *)
	MAIN_FAST.fbA26CH2.bRelay AT %QX44.5 : BOOL;	(*  ~ {LinkedWith:TIID^KG-HV A1 K-Bus [rechts]^KG-HV A1 (K-Bus)^KG-HV A26^Kanal 2^Ausgang} *)
	MAIN_FAST.fbA38OGCH1.bRelay AT %QX44.6 : BOOL;	(*  ~ {LinkedWith:TIID^KG-HV A1 K-Bus [rechts]^KG-HV A1 (K-Bus)^OG-UV A38^Kanal 1^Ausgang} *)
	MAIN_FAST.fbA38OGCH2.bRelay AT %QX44.7 : BOOL;	(*  ~ {LinkedWith:TIID^KG-HV A1 K-Bus [rechts]^KG-HV A1 (K-Bus)^OG-UV A38^Kanal 2^Ausgang} *)
	MAIN_FAST.fbA41OGCH1.bRelay AT %QX45.0 : BOOL;	(*  ~ {LinkedWith:TIID^KG-HV A1 K-Bus [rechts]^KG-HV A1 (K-Bus)^OG-UV A41^Kanal 1^OG-BadO Lampe} *)
	MAIN_FAST.fbA41OGCH2.bRelay AT %QX45.1 : BOOL;	(*  ~ {LinkedWith:TIID^KG-HV A1 K-Bus [rechts]^KG-HV A1 (K-Bus)^OG-UV A41^Kanal 2^Ausgang} *)
	MAIN_FAST.fbA43OGCH1.bRelay AT %QX45.2 : BOOL;	(*  ~ {LinkedWith:TIID^KG-HV A1 K-Bus [rechts]^KG-HV A1 (K-Bus)^OG-UV A43^Kanal 1^Ausgang} *)
	MAIN_FAST.fbA43OGCH2.bRelay AT %QX45.3 : BOOL;	(*  ~ {LinkedWith:TIID^KG-HV A1 K-Bus [rechts]^KG-HV A1 (K-Bus)^OG-UV A43^Kanal 2^Ausgang} *)
	MAIN_FAST.fbA44OGCH1.bRelay AT %QX45.4 : BOOL;	(*  ~ {LinkedWith:TIID^KG-HV A1 K-Bus [rechts]^KG-HV A1 (K-Bus)^OG-UV A44^Kanal 1^OG-KindN LampenWO} *)
	MAIN_FAST.fbA44OGCH2.bRelay AT %QX45.5 : BOOL;	(*  ~ {LinkedWith:TIID^KG-HV A1 K-Bus [rechts]^KG-HV A1 (K-Bus)^OG-UV A44^Kanal 2^OG-KindS LampenWO} *)
	MAIN_FAST.fbA45OGCH1.bRelay AT %QX45.6 : BOOL;	(*  ~ {LinkedWith:TIID^KG-HV A1 K-Bus [rechts]^KG-HV A1 (K-Bus)^OG-UV A45^Kanal 1^OG-KindN LampeM} *)
	MAIN_FAST.fbA45OGCH2.bRelay AT %QX45.7 : BOOL;	(*  ~ {LinkedWith:TIID^KG-HV A1 K-Bus [rechts]^KG-HV A1 (K-Bus)^OG-UV A45^Kanal 2^DG-KindO Lampe} *)
	MAIN_FAST.fbA48OGCH1.bRelay AT %QX46.0 : BOOL;	(*  ~ {LinkedWith:TIID^KG-HV A1 K-Bus [rechts]^KG-HV A1 (K-Bus)^OG-UV A48^Kanal 1^GaesteW LampenNS} *)
	MAIN_FAST.fbA48OGCH2.bRelay AT %QX46.1 : BOOL;	(*  ~ {LinkedWith:TIID^KG-HV A1 K-Bus [rechts]^KG-HV A1 (K-Bus)^OG-UV A48^Kanal 2^GaesteO LampenNS} *)
	MAIN_FAST.fbA49OGCH1.bRelay AT %QX46.2 : BOOL;	(*  ~ {LinkedWith:TIID^KG-HV A1 K-Bus [rechts]^KG-HV A1 (K-Bus)^OG-UV A49^Kanal 1^OG-BadDecke Lampen} *)
	MAIN_FAST.fbA49OGCH2.bRelay AT %QX46.3 : BOOL;	(*  ~ {LinkedWith:TIID^KG-HV A1 K-Bus [rechts]^KG-HV A1 (K-Bus)^OG-UV A49^Kanal 2^OG-BadON Lampe} *)
	MAIN_FAST.fbA50OGCH1.bRelay AT %QX46.4 : BOOL;	(*  ~ {LinkedWith:TIID^KG-HV A1 K-Bus [rechts]^KG-HV A1 (K-Bus)^OG-UV A50^Kanal 1^OG-WC Lampe} *)
	MAIN_FAST.fbA50OGCH2.bRelay AT %QX46.5 : BOOL;	(*  ~ {LinkedWith:TIID^KG-HV A1 K-Bus [rechts]^KG-HV A1 (K-Bus)^OG-UV A50^Kanal 2^Ausgang} *)
	MAIN_FAST.fbA52OGCH1.bRelay AT %QX46.6 : BOOL;	(*  ~ {LinkedWith:TIID^KG-HV A1 K-Bus [rechts]^KG-HV A1 (K-Bus)^OG-UV A52^Kanal 1^Ausgang} *)
	MAIN_FAST.fbA52OGCH2.bRelay AT %QX46.7 : BOOL;	(*  ~ {LinkedWith:TIID^KG-HV A1 K-Bus [rechts]^KG-HV A1 (K-Bus)^OG-UV A52^Kanal 2^Ausgang} *)
	MAIN_FAST.fbA53OGCH1.bRelay AT %QX47.0 : BOOL;	(*  ~ {LinkedWith:TIID^KG-HV A1 K-Bus [rechts]^KG-HV A1 (K-Bus)^OG-UV A53^Kanal 1^Balkon Steckdose} *)
	MAIN_FAST.fbA53OGCH2.bRelay AT %QX47.1 : BOOL;	(*  ~ {LinkedWith:TIID^KG-HV A1 K-Bus [rechts]^KG-HV A1 (K-Bus)^OG-UV A53^Kanal 2^Balkon Lampe} *)
	MAIN_FAST.fbA55OGCH1.bRelay AT %QX47.2 : BOOL;	(*  ~ {LinkedWith:TIID^KG-HV A1 K-Bus [rechts]^KG-HV A1 (K-Bus)^OG-UV A55^Kanal 1^AussenO Lampe} *)
	MAIN_FAST.fbA55OGCH2.bRelay AT %QX47.3 : BOOL;	(*  ~ {LinkedWith:TIID^KG-HV A1 K-Bus [rechts]^KG-HV A1 (K-Bus)^OG-UV A55^Kanal 2^AussenOS Lampe} *)
	MAIN_FAST.fbA56OGCH1.bRelay AT %QX47.4 : BOOL;	(*  ~ {LinkedWith:TIID^KG-HV A1 K-Bus [rechts]^KG-HV A1 (K-Bus)^OG-UV A56^Kanal 1^AussenWS Lampe} *)
	MAIN_FAST.fbA56OGCH2.bRelay AT %QX47.5 : BOOL;	(*  ~ {LinkedWith:TIID^KG-HV A1 K-Bus [rechts]^KG-HV A1 (K-Bus)^OG-UV A56^Kanal 2^AussenW Lampe} *)
	MAIN_FAST.fbA57OGCH1.bRelay AT %QX47.6 : BOOL;	(*  ~ {LinkedWith:TIID^KG-HV A1 K-Bus [rechts]^KG-HV A1 (K-Bus)^OG-UV A57^Kanal 1^AussenN Lampe} *)
	MAIN_FAST.fbA57OGCH2.bRelay AT %QX47.7 : BOOL;	(*  ~ {LinkedWith:TIID^KG-HV A1 K-Bus [rechts]^KG-HV A1 (K-Bus)^OG-UV A57^Kanal 2^Ausgang} *)
	MAIN_FAST.fbA15OGCH1.bRelay AT %QX48.0 : BOOL;	(*  ~ {LinkedWith:TIID^KG-HV A1 X001 EtherCAT [rechts]^OG-UV A1 Ethercat->K-Bus [unten links] ^OG-UV A15^Kanal 1^EssenNW Lampe} *)
	MAIN_FAST.fbA15OGCH2.bRelay AT %QX48.1 : BOOL;	(*  ~ {LinkedWith:TIID^KG-HV A1 X001 EtherCAT [rechts]^OG-UV A1 Ethercat->K-Bus [unten links] ^OG-UV A15^Kanal 2^Ausgang} *)
	MAIN_FAST.fbA17OGCH1.bRelay AT %QX48.2 : BOOL;	(*  ~ {LinkedWith:TIID^KG-HV A1 X001 EtherCAT [rechts]^OG-UV A1 Ethercat->K-Bus [unten links] ^OG-UV A17^Kanal 1^SchlafenO Lampe} *)
	MAIN_FAST.fbA17OGCH2.bRelay AT %QX48.3 : BOOL;	(*  ~ {LinkedWith:TIID^KG-HV A1 X001 EtherCAT [rechts]^OG-UV A1 Ethercat->K-Bus [unten links] ^OG-UV A17^Kanal 2^Ausgang} *)
	MAIN_FAST.fbA18OGCH1.bRelay AT %QX48.4 : BOOL;	(*  ~ {LinkedWith:TIID^KG-HV A1 X001 EtherCAT [rechts]^OG-UV A1 Ethercat->K-Bus [unten links] ^OG-UV A18^Kanal 1^WohnenSW Lampe} *)
	MAIN_FAST.fbA18OGCH2.bRelay AT %QX48.5 : BOOL;	(*  ~ {LinkedWith:TIID^KG-HV A1 X001 EtherCAT [rechts]^OG-UV A1 Ethercat->K-Bus [unten links] ^OG-UV A18^Kanal 2^WohnenM Beamer} *)
	MAIN_FAST.fbA19OGCH1.bRelay AT %QX48.6 : BOOL;	(*  ~ {LinkedWith:TIID^KG-HV A1 X001 EtherCAT [rechts]^OG-UV A1 Ethercat->K-Bus [unten links] ^OG-UV A19^Kanal 1^SchlafenWN Lampe} *)
	MAIN_FAST.fbA19OGCH2.bRelay AT %QX48.7 : BOOL;	(*  ~ {LinkedWith:TIID^KG-HV A1 X001 EtherCAT [rechts]^OG-UV A1 Ethercat->K-Bus [unten links] ^OG-UV A19^Kanal 2^SchlafenWM Lampe} *)
	MAIN_FAST.fbA21OGCH1.bRelay AT %QX49.0 : BOOL;	(*  ~ {LinkedWith:TIID^KG-HV A1 X001 EtherCAT [rechts]^OG-UV A1 Ethercat->K-Bus [unten links] ^OG-UV A21^Kanal 1^Ausgang} *)
	MAIN_FAST.fbA21OGCH2.bRelay AT %QX49.1 : BOOL;	(*  ~ {LinkedWith:TIID^KG-HV A1 X001 EtherCAT [rechts]^OG-UV A1 Ethercat->K-Bus [unten links] ^OG-UV A21^Kanal 2^Ausgang} *)
	MAIN_FAST.fbA23OGCH1.bRelay AT %QX49.2 : BOOL;	(*  ~ {LinkedWith:TIID^KG-HV A1 X001 EtherCAT [rechts]^OG-UV A1 Ethercat->K-Bus [unten links] ^OG-UV A23^Kanal 1^Ausgang} *)
	MAIN_FAST.fbA23OGCH2.bRelay AT %QX49.3 : BOOL;	(*  ~ {LinkedWith:TIID^KG-HV A1 X001 EtherCAT [rechts]^OG-UV A1 Ethercat->K-Bus [unten links] ^OG-UV A23^Kanal 2^Ausgang} *)
	MAIN_FAST.fbA25OGCH1.bRelay AT %QX49.4 : BOOL;	(*  ~ {LinkedWith:TIID^KG-HV A1 X001 EtherCAT [rechts]^OG-UV A1 Ethercat->K-Bus [unten links] ^OG-UV A25^Kanal 1^KochenO Lampen} *)
	MAIN_FAST.fbA25OGCH2.bRelay AT %QX49.5 : BOOL;	(*  ~ {LinkedWith:TIID^KG-HV A1 X001 EtherCAT [rechts]^OG-UV A1 Ethercat->K-Bus [unten links] ^OG-UV A25^Kanal 2^KochenN Lampe} *)
	MAIN_FAST.fbA26OGCH1.bRelay AT %QX49.6 : BOOL;	(*  ~ {LinkedWith:TIID^KG-HV A1 X001 EtherCAT [rechts]^OG-UV A1 Ethercat->K-Bus [unten links] ^OG-UV A26^Kanal 1^Speis Lampe} *)
	MAIN_FAST.fbA26OGCH2.bRelay AT %QX49.7 : BOOL;	(*  ~ {LinkedWith:TIID^KG-HV A1 X001 EtherCAT [rechts]^OG-UV A1 Ethercat->K-Bus [unten links] ^OG-UV A26^Kanal 2^EG-GangGarderobe Lampe} *)
	MAIN_FAST.fbA33OGCH1.bRelay AT %QX50.0 : BOOL;	(*  ~ {LinkedWith:TIID^KG-HV A1 X001 EtherCAT [rechts]^OG-UV A1 Ethercat->K-Bus [unten links] ^OG-UV A33^Kanal 1^EG-BadON Lampe} *)
	MAIN_FAST.fbA33OGCH2.bRelay AT %QX50.1 : BOOL;	(*  ~ {LinkedWith:TIID^KG-HV A1 X001 EtherCAT [rechts]^OG-UV A1 Ethercat->K-Bus [unten links] ^OG-UV A33^Kanal 2^Ausgang} *)
	MAIN_FAST.fbA35OGCH1.bRelay AT %QX50.2 : BOOL;	(*  ~ {LinkedWith:TIID^KG-HV A1 X001 EtherCAT [rechts]^OG-UV A1 Ethercat->K-Bus [unten links] ^OG-UV A35^Kanal 1^ArbeitenO Lampen} *)
	MAIN_FAST.fbA35OGCH2.bRelay AT %QX50.3 : BOOL;	(*  ~ {LinkedWith:TIID^KG-HV A1 X001 EtherCAT [rechts]^OG-UV A1 Ethercat->K-Bus [unten links] ^OG-UV A35^Kanal 2^ArbeitenW Lampen} *)
	MAIN_FAST.fbA36OGCH1.bRelay AT %QX50.4 : BOOL;	(*  ~ {LinkedWith:TIID^KG-HV A1 X001 EtherCAT [rechts]^OG-UV A1 Ethercat->K-Bus [unten links] ^OG-UV A36^Kanal 1^ArbeitenSO Steckdose} *)
	MAIN_FAST.fbA36OGCH2.bRelay AT %QX50.5 : BOOL;	(*  ~ {LinkedWith:TIID^KG-HV A1 X001 EtherCAT [rechts]^OG-UV A1 Ethercat->K-Bus [unten links] ^OG-UV A36^Kanal 2^Ausgang} *)
	MAIN_FAST.fbA78OGCH1.bRelay AT %QX50.6 : BOOL;	(*  ~ {LinkedWith:TIID^KG-HV A1 K-Bus [rechts]^KG-HV A1 (K-Bus)^OG-UV A78^Kanal 1^Ausgang} *)
	MAIN_FAST.fbA78OGCH2.bRelay AT %QX50.7 : BOOL;	(*  ~ {LinkedWith:TIID^KG-HV A1 K-Bus [rechts]^KG-HV A1 (K-Bus)^OG-UV A78^Kanal 2^Dachboden Lampe} *)
	MAIN_FAST.fbA80OGCH1.bRelay AT %QX51.0 : BOOL;	(*  ~ {LinkedWith:TIID^KG-HV A1 K-Bus [rechts]^KG-HV A1 (K-Bus)^OG-UV A80 (reserve)^Kanal 1^Ausgang} *)
	MAIN_FAST.fbA80OGCH2.bRelay AT %QX51.1 : BOOL;	(*  ~ {LinkedWith:TIID^KG-HV A1 K-Bus [rechts]^KG-HV A1 (K-Bus)^OG-UV A80 (reserve)^Kanal 2^Ausgang} *)
END_VAR

(* Data type *)
TYPE Baudrate: (
	B300    :=  1,   (*               EL6002        EL6022 *)
	B600    :=  2,   (*               EL6002        EL6022 *)
	B1200   :=  3,   (*               EL6002        EL6022 *)
	B2400   :=  4,   (* EL6001        EL6002 EL6021 EL6022 *)
	B4800   :=  5,   (* EL6001        EL6002 EL6021 EL6022 *)
	B9600   :=  6,   (* EL6001        EL6002 EL6021 EL6022 *)
	B12000  := 14,   (* EL6001 FW>=07                      *)
	B14400  := 15,   (* EL6001 FW>=07                      *)
	B19200  :=  7,   (* EL6001        EL6002 EL6021 EL6022 *)
	B38400  :=  8,   (* EL6001        EL6002 EL6021 EL6022 *)
	B57600  :=  9,   (* EL6001        EL6002 EL6021 EL6022 *)
	B115200 := 10    (* EL6001        EL6002 EL6021 EL6022 *)
);
END_TYPE

(* Data type *)
TYPE Dataframe : (
	FMT_7E1 :=  1,   (* EL6001 EL6021 *)
	FMT_7O1 :=  2,   (* EL6001 EL6021 *)
	FMT_8N1 :=  3,   (* EL6001 EL6021 *)
	FMT_8E1 :=  4,   (* EL6001 EL6021 *)
	FMT_8O1 :=  5,   (* EL6001 EL6021 *)
	FMT_7N2 :=  8,   (*               EL6002 FW>=03*)
	FMT_7E2 :=  9,   (* EL6001 EL6021 *)
	FMT_7O2 := 10,   (* EL6001 EL6021 *)
	FMT_8N2 := 11,   (* EL6001 EL6021 *)
	FMT_8E2 := 12,   (* EL6001 EL6021 *)
	FMT_8O2 := 13    (* EL6001 EL6021 *)
);
END_TYPE

(* Data type *)
TYPE E_FroelingAnlagenzustand : (
	Winterbetrieb := 0,
	Sommerbetrieb := 1,
	Uebergangsbetrieb := 2,
	KeinScheitholzbetrieb := 3,
	Ausgeschaltet := 5,
	Extraheizen := 6,
	Kaminkehrer := 7,
	Reinigen := 8
);
END_TYPE

(* Data type *)
TYPE E_FroelingKesselzustand : (
	Stoerung := 0,
	KesselAus := 1,
	Anheizen := 2,
	Heizen := 3,
	Feuererhaltung := 4,
	FeuerAus := 5,
	TuerOffen := 6,
	Vorbereitung := 7,
	Vorwaermen := 8,
	Zuenden := 9,
	AbstellenWarten := 10,
	AbstellenWarten1 := 11,
	AbstellenEinschub1 := 12,
	AbstellenWarten2 := 13,
	AbstellenEinschub2 := 14,
	Abreinigen := 15,
	Warten2h := 16,
	Saugen_Heizen := 17,
	Fehlzuendung := 18,
	Betriebsbereit := 19,
	RostSchliessen := 20,
	StokerLeeren := 21,
	Vorheizen := 22,
	Saugen := 23,
	RseSchliessen := 24,
	RseOeffnen := 25,
	RostKippen := 26,
	Vorwaermen_Zuenden := 27,
	Resteinschub := 28,
	StokerAuffuellen := 29,
	LambdasondeAufheizen := 30,
	GeblaesenachlaufI := 31,
	GeblaesenachlaufII := 32,
	Abgestellt := 33,
	NachZuenden := 34,
	ZuendenWarten := 35,
	Fehlerbehebung20min := 66,
	ReinigenMoeglich := 69
);
END_TYPE

(* Data type *)
TYPE E_ModbusFunction : (
	ReadCoils := 1,
	ReadInputStatus := 2,
	ReadRegs := 3,
	ReadInputRegs := 4,
	WriteSingleCoil := 5,
	WriteSingleRegister := 6,
	Diagnostics := 8,
	WriteMultipleCoils := 15,
	WriteRegs := 16
);
END_TYPE

(* Data type *)
TYPE E_TemperatureUnit : (
	KELVIN,
	GRAD_CELSIUS,
	GRAD_FAHRENHEIT,
	GRAD_RANKINE,
	GRAD_DELISLE,
	GRAD_REAUMUR,
	GRAD_NEWTON,
	GRAD_ROMER
);
END_TYPE

(* Data type *)
TYPE ST_ModbusAddressRange :
STRUCT
	start: UINT;
	length: UINT;
	accessFunction: E_ModbusFunction;
END_STRUCT
END_TYPE

(* Data type *)
TYPE ST_TemperatureUnit :
STRUCT
	id: E_TemperatureUnit;
	unit: STRING;
	symbol: STRING;
	f1: REAL;
	f2: REAL;
	offset: REAL;
	scale: REAL;
	inventor: STRING;
END_STRUCT
END_TYPE

(* Data type *)
TYPE stDeviceSpace :
STRUCT
	byModbusSlaveAddress : BYTE;
	wModbusAdress : WORD;
	iModbusFunction : INT;
	pSPSDataSpace : DWORD;
	wSPSDataSpaceLength : WORD;
END_STRUCT
END_TYPE

(* Data type *)
TYPE stFB_ModbusMaster :
STRUCT
	byCurrentModbusSlaveAdress: BYTE;
	bModbusAddressExist: BOOL;
	bModbusCommunicationActive: BOOL;
	stCurrentDeviceSpace:  ARRAY [0..uiMaxCurrentDeviceSpace] OF stDeviceSpace;
	iNumberOfData: INT;
	bError: BOOL;
	eError: INT;
END_STRUCT
END_TYPE

(* Data type *)
TYPE stResultOfModbusSlaveScan :
STRUCT
	eModbusfunction: MODBUS_FUNCTIONS;
	iModbusAdress: INT;
	wValue: WORD;
	eModbusError: MODBUS_ERRORS;
END_STRUCT
END_TYPE

(* POU MAIN, ST *)
PROGRAM MAIN
VAR CONSTANT
	JALOUSIE_UD_TIME_TERASSE: TIME := t#35s500ms;
	JALOUSIE_UD_TIME_BALKON: TIME := t#35s500ms;
	JALOUSIE_UD_TIME_WINDOW_EG: TIME := t#35s500ms;
	JALOUSIE_UD_TIME_WINDOW_OG: TIME := t#37s500ms;
END_VAR
VAR
	ups: FB_S_UPS;
(*sensoren*)
	_bwmAussenW        AT %I*: BOOL; (* West *)
	_bwmAussenSO       AT %I*: BOOL; (* Sued-Ost *)
	_bwmEgGang         AT %I*: BOOL; (* Sued *)
	_bwmEgWc           AT %I*: BOOL; (* Sued-West *)
	_bwmHobby          AT %I*: BOOL; (* Sued-West *)
	_bwmKgGang         AT %I*: BOOL; (* Ost *)
	_bwmKochen         AT %I*: BOOL; (* Sued-West *)
	_bwmLager          AT %I*: BOOL; (* Sued-West *)
	_bwmOgGang         AT %I*: BOOL; (* Sued-West *)
	_bwmWaschen        AT %I*: BOOL; (* Ost *)
	_lichtEgGang_status  AT %I*: USINT;
	_lichtEgGang_dataIn  AT %I*: INT;
	_lichtEgWc_status    AT %I*: USINT;
	_lichtEgWc_dataIn    AT %I*: INT;
	_lichtHobby_status   AT %I*: USINT;
	_lichtHobby_dataIn   AT %I*: INT;
	_lichtKochen_status  AT %I*: USINT;
	_lichtKochen_dataIn  AT %I*: INT;
	_lichtLager_status   AT %I*: USINT;
	_lichtLager_dataIn   AT %I*: INT;
	_lichtOgGang_status  AT %I*: USINT;
	_lichtOgGang_dataIn  AT %I*: INT;
	_lichtWaschen_status AT %I*: USINT;
	_lichtWaschen_dataIn AT %I*: INT;
	_temperaturArbeiten_status AT %I*: USINT;
	_temperaturArbeiten_dataIn AT %I*: INT;
	_temperaturEgBad_status AT %I*: USINT;
	_temperaturEgBad_dataIn AT %I*: INT;
	_temperaturEgGangSM_status AT %I*: USINT;
	_temperaturEgGangSM_dataIn AT %I*: INT;
	_temperaturEgGangSO_status AT %I*: USINT;
	_temperaturEgGangSO_dataIn AT %I*: INT;
	_temperaturEgWc_status AT %I*: USINT;
	_temperaturEgWc_dataIn AT %I*: INT;
	_temperaturEssen_status AT %I*: USINT;
	_temperaturEssen_dataIn AT %I*: INT;
	_temperaturGaeste_status AT %I*: USINT;
	_temperaturGaeste_dataIn AT %I*: INT;
	_temperaturHobby_status AT %I*: USINT;
	_temperaturHobby_dataIn AT %I*: INT;
	_temperaturKochen_status AT %I*: USINT;
	_temperaturKochen_dataIn AT %I*: INT;
	_temperaturLager_status AT %I*: USINT;
	_temperaturLager_dataIn AT %I*: INT;
	_temperaturOgBad_status AT %I*: USINT;
	_temperaturOgBad_dataIn AT %I*: INT;
	_temperaturOgGang_status AT %I*: USINT;
	_temperaturOgGang_dataIn AT %I*: INT;
	_temperaturOgKind_status AT %I*: USINT;
	_temperaturOgKind_dataIn AT %I*: INT;
	_temperaturOgWc_status AT %I*: USINT;
	_temperaturOgWc_dataIn AT %I*: INT;
	_temperaturSchlafen_status AT %I*: USINT;
	_temperaturSchlafen_dataIn AT %I*: INT;
	_temperaturVorrat_status AT %I*: USINT;
	_temperaturVorrat_dataIn AT %I*: INT;
	_temperaturWaschenON_status AT %I*: USINT;
	_temperaturWaschenON_dataIn AT %I*: INT;
	_temperaturWaschenOS_status AT %I*: USINT;
	_temperaturWaschenOS_dataIn AT %I*: INT;
	_temperaturWohnen_status AT %I*: USINT;
	_temperaturWohnen_dataIn AT %I*: INT;
	_tasterArbeitenOO  AT %I*: BOOL; (* Ost *)
	_tasterArbeitenOL  AT %I*: BOOL; (* Ost *)
	_tasterArbeitenOR  AT %I*: BOOL; (* Ost *)
	_tasterArbeitenSL  AT %I*: BOOL; (* Sued *)
	_tasterArbeitenSR  AT %I*: BOOL; (* Sued *)
	_tasterDgKind      AT %I*: BOOL; (* West-Sued *)
	_tasterEgBadL      AT %I*: BOOL; (* Sued *)
	_tasterEgBadR      AT %I*: BOOL; (* Sued *)
	_tasterEgGang      AT %I*: BOOL; (* Nord-West *)
	_tasterEgWc        AT %I*: BOOL; (* West-Nord *)
	_tasterEssenO      AT %I*: BOOL; (* Nord *)
	_tasterEssenL      AT %I*: BOOL; (* Nord *)
	_tasterEssenR      AT %I*: BOOL; (* Nord *)
	_tasterGaesteO     AT %I*: BOOL; (* Nord *)
	_tasterGaesteL     AT %I*: BOOL; (* Nord *)
	_tasterGaesteR     AT %I*: BOOL; (* Nord *)
	_tasterHeizen      AT %I*: BOOL; (* Sued-West *)
	_tasterHobbyL      AT %I*: BOOL; (* Ost *)
	_tasterHobbyR      AT %I*: BOOL; (* Ost *)
	_tasterKochenOL    AT %I*: BOOL; (* Ost *)
	_tasterKochenOR    AT %I*: BOOL; (* Ost *)
	_tasterKochenWO    AT %I*: BOOL; (* West *)
	_tasterKochenWL    AT %I*: BOOL; (* West *)
	_tasterKochenWR    AT %I*: BOOL; (* West *)
	_tasterLagerNO     AT %I*: BOOL; (* Nord-Ost *)
	_tasterLagerS      AT %I*: BOOL; (* Sued *)
	_tasterOgBadL      AT %I*: BOOL; (* Sued *)
	_tasterOgBadR      AT %I*: BOOL; (* Sued *)
	_tasterOgKindNO    AT %I*: BOOL; (* Nord *)
	_tasterOgKindNL    AT %I*: BOOL; (* Nord *)
	_tasterOgKindNR    AT %I*: BOOL; (* Nord *)
	_tasterOgKindWL    AT %I*: BOOL; (* West *)
	_tasterOgKindWR    AT %I*: BOOL; (* West *)
	_tasterOgWc        AT %I*: BOOL; (* West *)
	_tasterSchlafenOo  AT %I*: BOOL; (* Ost *)
	_tasterSchlafenOl  AT %I*: BOOL; (* Ost *)
	_tasterSchlafenOr  AT %I*: BOOL; (* Ost *)
	_tasterSchlafenWML AT %I*: BOOL; (* West-Mitte *)
	_tasterSchlafenWMR AT %I*: BOOL; (* West-Mitte *)
	_tasterSchlafenWNL AT %I*: BOOL; (* West-Nord *)
	_tasterSchlafenWNR AT %I*: BOOL; (* West-Nord *)
	_tasterSpeis       AT %I*: BOOL; (* Tuerkontakt *)
	_tasterWaschenL    AT %I*: BOOL; (* West-Sued *)
	_tasterWaschenR    AT %I*: BOOL; (* West-Sued *)
	_tasterWohnenOO    AT %I*: BOOL; (* Ost *)
	_tasterWohnenOL    AT %I*: BOOL; (* Ost *)
	_tasterWohnenOR    AT %I*: BOOL; (* Ost *)
	_tasterWohnenWO    AT %I*: BOOL; (* West *)
	_tasterWohnenWL    AT %I*: BOOL; (* West *)
	_tasterWohnenWR    AT %I*: BOOL; (* West *)
(*aktoren*)
	_dimmerWohnenN_intensity AT %I*: REAL := 67;
	_dimmerWohnenN_status    AT %I*: USINT;
	_dimmerWohnenN_dataIn    AT %I*: INT;
	_dimmerWohnenN_dataOut   AT %Q*: INT;
	_dimmerWohnenN_control   AT %Q*: USINT;
	_dimmerEgBadSM_intensity AT %I*: REAL := 67;
	_dimmerEgBadSM_status    AT %I*: USINT;
	_dimmerEgBadSM_dataIn    AT %I*: INT;
	_dimmerEgBadSM_dataOut   AT %Q*: INT;
	_dimmerEgBadSM_control   AT %Q*: USINT;
	_lampeEgBadOM      AT %Q*: BOOL; (* Ost (Spiegel) *)
	_lampeEgGang       AT %Q*: BOOL; (* Sued *)
	_lampeEgWc         AT %Q*: BOOL; (* West *)
	_lampeEssenM       AT %Q*: BOOL; (* Mitte *)
	_lampeEssenS       AT %Q*: BOOL; (* Sued *)
	_lampeKochenSW     AT %Q*: BOOL; (* Sued-West *)
	_lampeOgGang       AT %Q*: BOOL; (* 3 *)
	_lampeEgOgStiege   AT %Q*: BOOL; (* Ost *)
	_lampeSchlafenS    AT %Q*: BOOL; (* Sued-West | Sued-Ost*)
	_lampeWohnenM      AT %Q*: BOOL; (* Mitte *)

(* KG *)

	heizenTaster: FB_Button;
	heizenLampe:  FB_Lamp;
	heizenHK1:    FB_Heizkreis;
	heizenHK2:    FB_Heizkreis;

	hobbyBwm: FB_Motion;
	hobbyLicht: FB_Light;
	hobbyTasterL: FB_Button;
	hobbyTasterR: FB_Button;
	hobbyTemperatur: FB_Temperature;
	hobbyLampeN: FB_Lamp;
	hobbyLampeS: FB_Lamp;

	lagerBwm: FB_Motion;
	lagerLicht: FB_Light;
	lagerTasterNO: FB_Button;
	lagerTasterS: FB_Button;
	lagerTemperatur: FB_Temperature;
	lagerLampe: FB_Lamp;

	vorratTemperatur: FB_Temperature;
	vorratLampe: FB_Lamp;

	waschenBwm: FB_Motion;
	waschenLicht: FB_Light;
	waschenTasterL: FB_Button;
	waschenTasterR: FB_Button;
	waschenTemperaturON: FB_Temperature;
	waschenTemperaturOS: FB_Temperature;
	waschenLampeNM: FB_Lamp;
	waschenLampeS: FB_Lamp;

	kgGangBwm: FB_Motion;
	kgGangLampe: FB_Lamp;

	kgEgLampe: FB_Lamp;

(* EG *)

	egBadTasterR:    FB_Button;
	egBadTasterL:    FB_Button;
	egBadTemperatur: FB_Temperature;
	egBadDimmerSM:   FB_Dimmer;
	egBadLampeON:    FB_Lamp;
	egBadLampeOM:    FB_Lamp;
	egBadLampeSM:    FB_Lamp;
	egBadJalousie:   FB_Jalousie;

	egGangBwm:          FB_Motion;
	egGangLicht:        FB_Light;
	egGangTaster:       FB_Button;
	egGangTemperaturSM: FB_Temperature;
	egGangTemperaturSO: FB_Temperature;
	egGangLampe:        FB_Lamp;

	egWcBwm:        FB_Motion;
	egWcLicht:      FB_Light;
	egWcTaster:     FB_Button;
	egWcTemperatur: FB_Temperature;
	egWcLampe:      FB_Lamp;

	essenTasterO:    FB_Button;
	essenTasterL:    FB_Button;
	essenTasterR:    FB_Button;
	essenTemperatur: FB_Temperature;
	essenLampeS:     FB_Lamp;
	essenLampeM:     FB_Lamp;
	essenLampeNW:    FB_Lamp;
	essenJalousie:   FB_Jalousie;

	kochenBwm:        FB_Motion;
	kochenLicht:      FB_Light;
	kochenTasterOL:   FB_Button;
	kochenTasterOR:   FB_Button;
	kochenTasterWO:   FB_Button;
	kochenTasterWL:   FB_Button;
	kochenTasterWR:   FB_Button;
	kochenTemperatur: FB_Temperature;
	kochenLampeO:     FB_Lamp;
	kochenLampeN:     FB_Lamp;
	kochenLampeSW:    FB_Lamp;
	kochenJalousieS:  FB_Jalousie;
	kochenJalousieO:  FB_Jalousie;

	schlafenTasterOo:   FB_Button;
	schlafenTasterOl:   FB_Button;
	schlafenTasterOr:   FB_Button;
	schlafenTasterWML:  FB_Button;
	schlafenTasterWMR:  FB_Button;
	schlafenTasterWNL:  FB_Button;
	schlafenTasterWNR:  FB_Button;
	schlafenTemperatur: FB_Temperature;
	schlafenLampeS:     FB_Lamp;
	schlafenLampeO:     FB_Lamp;
	schlafenLampeWM:    FB_Lamp;
	schlafenLampeWN:    FB_Lamp;
	schlafenJalousieN:  FB_Jalousie;
	schlafenJalousieW:  FB_Jalousie;

	speisTuer:  FB_Button;
	speisLampe: FB_Lamp;

	wohnenTasterOO:   FB_Button;
	wohnenTasterOR:   FB_Button;
	wohnenTasterOL:   FB_Button;
	wohnenTasterWO:   FB_Button;
	wohnenTasterWR:   FB_Button;
	wohnenTasterWL:   FB_Button;
	wohnenTemperatur: FB_Temperature;
	wohnenLampeM:     FB_Lamp;
	wohnenLampeN:     FB_Lamp;
	wohnenLampeSW:    FB_Lamp;
	wohnenDimmerN:    FB_Dimmer;
	wohnenJalousieS:  FB_Jalousie;
	wohnenJalousieWa: FB_Jalousie;
	wohnenJalousieWb: FB_Jalousie;

	egOgLampe: FB_Lamp;

(* OG *)

	arbeitenTemperatur: FB_Temperature;
	arbeitenTasterOO:   FB_Button;
	arbeitenTasterOL:   FB_Button;
	arbeitenTasterOR:   FB_Button;
	arbeitenTasterSL:   FB_Button;
	arbeitenTasterSR:   FB_Button;
	arbeitenLampeN:     FB_Lamp;
	arbeitenLampeS:     FB_Lamp;
	arbeitenLampeSW:    FB_Lamp;
	arbeitenJalousieN:  FB_Jalousie;
	arbeitenJalousieW:  FB_Jalousie;
	arbeitenJalousieS:  FB_Jalousie;

	gaesteTasterO:    FB_Button;
	gaesteTasterR:    FB_Button;
	gaesteTasterL:    FB_Button;
	gaesteTemperatur: FB_Temperature;
	gaesteLampeO:     FB_Lamp;
	gaesteLampeW:     FB_Lamp;
	gaesteJalousieO:  FB_Jalousie;
	gaesteJalousieS:  FB_Jalousie;

	ogBadTasterR:    FB_Button;
	ogBadTasterL:    FB_Button;
	ogBadTemperatur: FB_Temperature;
	ogBadLampeON:    FB_Lamp;
	ogBadLampeOM:    FB_Lamp;
	ogBadLampeSM:    FB_Lamp;
	ogBadJalousie:   FB_Jalousie;

	ogGangBwm:        FB_Motion;
	ogGangLicht:      FB_Light;
	ogGangTemperatur: FB_Temperature;
	ogGangLampe:      FB_Lamp;

	ogKindTasterNO:   FB_Button;
	ogKindTasterNR:   FB_Button;
	ogKindTasterNL:   FB_Button;
	ogKindTasterWR:   FB_Button;
	ogKindTasterWL:   FB_Button;
	ogKindTemperatur: FB_Temperature;
	ogKindLampeN:     FB_Lamp;
	ogKindLampeM:     FB_Lamp;
	ogKindLampeS:     FB_Lamp;
	ogKindJalousieS:  FB_Jalousie;
	ogKindJalousieW:  FB_Jalousie;

	ogWcTaster:     FB_Button;
	ogWcTemperatur: FB_Temperature;
	ogWcLampe:      FB_Lamp;

(* DG *)

	dgKindTaster:     FB_Button;
	dachbodenLampe:   FB_Lamp;
	dgKindLampe:      FB_Lamp;

(* Aussen *)

	aussenBwmW:  FB_Motion;
	aussenBwmSO: FB_Motion;
END_VAR
ups();

(* input processing *)

aussenBwmW(IN := _bwmAussenW, ROOM := 'Aussen', LOCATION := 'West');
aussenBwmSO(IN := _bwmAussenSO, ROOM := 'Aussen', LOCATION := 'Sued-Ost');
kgGangBwm(IN := _bwmKgGang, ROOM := 'KG-Gang', LOCATION := 'Ost');
heizenTaster(IN := _tasterHeizen, ROOM := 'Heizen', LOCATION := 'Nord-West');
hobbyBwm(IN := _bwmHobby, ROOM := 'Hobby', LOCATION := 'Sued-West');
hobbyLicht(Status := _lichtHobby_status, DataIn := _lichtHobby_dataIn, ROOM := 'Hobby', LOCATION := 'Sued-West');
hobbyTasterL(IN := _tasterHobbyL, ROOM := 'Hobby', LOCATION := 'Ost');
hobbyTasterR(IN := _tasterHobbyR, ROOM := 'Hobby', LOCATION := 'Ost');
lagerBwm(IN := _bwmLager, ROOM := 'Lager', LOCATION := 'Sued-West');
lagerLicht(Status := _lichtLager_status, DataIn := _lichtLager_dataIn, ROOM := 'Lager', LOCATION := 'Sued-West');
lagerTasterNO(IN := _tasterLagerNO, ROOM := 'Lager', LOCATION := 'Nord-Ost');
lagerTasterS(IN := _tasterLagerS, ROOM := 'Lager', LOCATION := 'Sued');
vorratTemperatur(Status := _temperaturVorrat_status, DataIn := _temperaturVorrat_dataIn,
	ROOM := 'Vorrat', LOCATION := 'Sued-West');
waschenBwm(IN := _bwmWaschen, ROOM := 'Waschen', LOCATION := 'Ost');
waschenLicht(Status := _lichtWaschen_status, DataIn := _lichtWaschen_dataIn, ROOM := 'Lager', LOCATION := 'Sued-West');
waschenTasterL(IN := _tasterWaschenL, ROOM := 'Waschen', LOCATION := 'West-Sued');
waschenTasterR(IN := _tasterWaschenR, ROOM := 'Waschen', LOCATION := 'West-Sued');
waschenTemperaturON(Status := _temperaturWaschenON_status, DataIn := _temperaturWaschenON_dataIn,
	ROOM := 'Vorrat', LOCATION := 'Sued-West');

egBadTasterL(IN := _tasterEgBadL, ROOM := 'EG-Bad', LOCATION := 'Sued');
egBadTasterR(IN := _tasterEgBadR, ROOM := 'EG-Bad', LOCATION := 'Sued');
egBadTemperatur(Status := _temperaturEgBad_status, DataIn := _temperaturEgBad_dataIn,
	ROOM := 'EG-Bad', LOCATION := 'Sued-Ost');
egGangBwm(IN := _bwmEgGang, ROOM := 'EG-Gang', LOCATION := 'Sued');
egGangLicht(Status := _lichtEgGang_status, DataIn := _lichtEgGang_dataIn, ROOM := 'EG-Gang', Location := 'Sued');
egGangTaster(IN := _tasterEgGang, ROOM := 'EG-Gang', LOCATION := 'Nord-West');
egGangTemperaturSM(Status := _temperaturEgGangSM_status, DataIn := _temperaturEgGangSM_dataIn,
	ROOM := 'EG-Gang', LOCATION := 'Sued-Mitte');
egWcBwm(IN := _bwmEgWc, ROOM := 'EG-WC', LOCATION := 'Sued-West');
egWcLicht(Status := _lichtEgWc_status, DataIn := _lichtEgWc_dataIn, ROOM := 'EG-WC', Location := 'Sued-West');
egWcTaster(IN := _tasterEgWc, ROOM := 'EG-WC', LOCATION := 'West-Sued');
essenTasterO(IN := _tasterEssenO, ROOM := 'Essen', LOCATION := 'Nord');
essenTasterL(IN := _tasterEssenL, ROOM := 'Essen', LOCATION := 'Nord');
essenTasterR(IN := _tasterEssenR, ROOM := 'Essen', LOCATION := 'Nord');
essenTemperatur(Status := _temperaturEssen_status, DataIn := _temperaturEssen_dataIn,
	ROOM := 'Essen', LOCATION := 'Sued-West');
kochenBwm(IN := _bwmKochen, ROOM := 'Kochen', LOCATION := 'Sued-West');
kochenLicht(Status := _lichtKochen_status, DataIn := _lichtKochen_dataIn, ROOM := 'Kochen', Location := 'Sued-West');
kochenTasterWO(IN := _tasterKochenWO, ROOM := 'Kochen', Location := 'West');
kochenTasterWL(IN := _tasterKochenWL, ROOM := 'Kochen', Location := 'West');
kochenTasterWR(IN := _tasterKochenWR, ROOM := 'Kochen', Location := 'West');
kochenTasterOL(IN := _tasterKochenOL, ROOM := 'Kochen', Location := 'Ost');
kochenTasterOR(IN := _tasterKochenOR, ROOM := 'Kochen', Location := 'Ost');
kochenTemperatur(Status := _temperaturKochen_status, DataIn := _temperaturKochen_dataIn,
	ROOM := 'Kochen', LOCATION := 'Sued-West');
schlafenTasterWML(IN := _tasterSchlafenWML, ROOM := 'Schlafen', LOCATION := 'West-Mitte');
schlafenTasterWMR(IN := _tasterSchlafenWMR, ROOM := 'Schlafen', LOCATION := 'West-Mitte');
schlafenTasterWNL(IN := _tasterSchlafenWNL, ROOM := 'Schlafen', LOCATION := 'West-Nord');
schlafenTasterWNR(IN := _tasterSchlafenWNR, ROOM := 'Schlafen', LOCATION := 'West-Nord');
schlafenTasterOo(IN := _tasterSchlafenOo, ROOM := 'Schlafen', LOCATION := 'Ost');
schlafenTasterOl(IN := _tasterSchlafenOl, ROOM := 'Schlafen', LOCATION := 'Ost');
schlafenTasterOr(IN := _tasterSchlafenOr, ROOM := 'Schlafen', LOCATION := 'Ost');
schlafenTemperatur(Status := _temperaturSchlafen_status, DataIn := _temperaturSchlafen_dataIn,
	ROOM := 'Schlafen', LOCATION := 'Nord-West');
speisTuer(IN := _tasterSpeis, ROOM := 'Speis', LOCATION := 'Tuerkontakt');
wohnenTasterOO(IN := _tasterWohnenOO, ROOM := 'Wohnen', LOCATION := 'Ost');
wohnenTasterOL(IN := _tasterWohnenOL, ROOM := 'Wohnen', LOCATION := 'Ost');
wohnenTasterOR(IN := _tasterWohnenOR, ROOM := 'Wohnen', LOCATION := 'Ost');
wohnenTasterWO(IN := _tasterWohnenWO, ROOM := 'Wohnen', LOCATION := 'West');
wohnenTasterWL(IN := _tasterWohnenWL, ROOM := 'Wohnen', LOCATION := 'West');
wohnenTasterWR(IN := _tasterWohnenWR, ROOM := 'Wohnen', LOCATION := 'West');
wohnenTemperatur(Status := _temperaturWohnen_status, DataIn := _temperaturWohnen_dataIn,
	ROOM := 'Wohnen', LOCATION := 'Sued-West');

arbeitenTasterOO(IN := _tasterArbeitenOO, ROOM := 'Arbeiten', LOCATION := 'Ost');
arbeitenTasterOL(IN := _tasterArbeitenOL, ROOM := 'Arbeiten', LOCATION := 'Ost');
arbeitenTasterOR(IN := _tasterArbeitenOR, ROOM := 'Arbeiten', LOCATION := 'Ost');
arbeitenTasterSL(IN := _tasterArbeitenSL, ROOM := 'Arbeiten', LOCATION := 'Sued');
arbeitenTasterSR(IN := _tasterArbeitenSR, ROOM := 'Arbeiten', LOCATION := 'Sued');
arbeitenTemperatur(Status := _temperaturArbeiten_status, DataIn := _temperaturArbeiten_dataIn,
	ROOM := 'Arbeiten', LOCATION := 'Nord-Ost');
gaesteTasterO(IN := _tasterGaesteO, ROOM := 'Gaeste', LOCATION := 'Nord');
gaesteTasterL(IN := _tasterGaesteL, ROOM := 'Gaeste', LOCATION := 'Nord');
gaesteTasterR(IN := _tasterGaesteR, ROOM := 'Gaeste', LOCATION := 'Nord');
gaesteTemperatur(Status := _temperaturGaeste_status, DataIn := _temperaturGaeste_dataIn,
	ROOM := 'Gaeste', LOCATION := 'Ost-Nord');
ogKindTasterNO(IN := _tasterOgKindNO, ROOM := 'OG-Kind', LOCATION := 'Nord');
ogKindTasterNL(IN := _tasterOgKindNL, ROOM := 'OG-Kind', LOCATION := 'Nord');
ogKindTasterNR(IN := _tasterOgKindNR, ROOM := 'OG-Kind', LOCATION := 'Nord');
ogKindTasterWL(IN := _tasterOgKindWL, ROOM := 'OG-Kind', LOCATION := 'West');
ogKindTasterWR(IN := _tasterOgKindWR, ROOM := 'OG-Kind', LOCATION := 'West');
ogKindTemperatur(Status := _temperaturOgKind_status, DataIn := _temperaturOgKind_dataIn,
	ROOM := 'OG-Kind', LOCATION := 'Ost-Nord');
ogBadTasterL(IN := _tasterOgBadL, ROOM := 'OG-Bad', LOCATION := 'Sued');
ogBadTasterR(IN := _tasterOgBadR, ROOM := 'OG-Bad', LOCATION := 'Sued');
ogBadTemperatur(Status := _temperaturOgBad_status, DataIn := _temperaturOgBad_dataIn,
	ROOM := 'OG-Bad', LOCATION := 'Sued-Ost');
ogGangBwm(IN := _bwmOgGang, ROOM := 'OG-Gang', LOCATION := 'Sued-West');
ogGangLicht(ROOM := 'OG-Gang', LOCATION := 'Sued-West');
ogGangTemperatur(Status := _temperaturOgGang_status, DataIn := _temperaturOgGang_dataIn,
	ROOM := 'OG-Gang', LOCATION := 'Sued-West');
ogWcTaster(IN := _tasterOgWc, ROOM := 'OG-WC', LOCATION := 'Ost-Sued');
ogWcTemperatur(Status := _temperaturOgWc_status, DataIn := _temperaturOgWc_dataIn,
	ROOM := 'OG-WC', LOCATION := 'Ost-Sued');

dgKindTaster(IN := _tasterDgKind, Room := 'DG-Kind', LOCATION := 'West-Sued');

(* control *)

arbeitenJalousieN(T_UD := JALOUSIE_UD_TIME_WINDOW_OG, T_ANGLE:= t#1s);
arbeitenJalousieW(T_UD := JALOUSIE_UD_TIME_WINDOW_OG, T_ANGLE:= t#1s);
arbeitenJalousieS(T_UD := JALOUSIE_UD_TIME_BALKON, T_ANGLE:= t#1s);
egBadJalousie(T_UD := JALOUSIE_UD_TIME_WINDOW_EG, T_ANGLE:= t#1s);
essenJalousie(T_UD := JALOUSIE_UD_TIME_WINDOW_EG, T_ANGLE:= t#1s);
gaesteJalousieS(T_UD := JALOUSIE_UD_TIME_WINDOW_OG, T_ANGLE:= t#1s);
gaesteJalousieO(T_UD := JALOUSIE_UD_TIME_WINDOW_OG, T_ANGLE:= t#1s);
kochenJalousieS(T_UD := JALOUSIE_UD_TIME_WINDOW_EG, T_ANGLE:= t#1s);
kochenJalousieO(T_UD := JALOUSIE_UD_TIME_WINDOW_EG, T_ANGLE:= t#1s);
ogBadJalousie(T_UD := JALOUSIE_UD_TIME_WINDOW_OG, T_ANGLE:= t#1s);
ogKindJalousieW(T_UD := JALOUSIE_UD_TIME_BALKON, T_ANGLE:= t#1s);
ogKindJalousieS(T_UD := JALOUSIE_UD_TIME_WINDOW_OG, T_ANGLE:= t#1s);
schlafenJalousieN(T_UD := JALOUSIE_UD_TIME_WINDOW_EG, T_ANGLE:= t#1s);
schlafenJalousieW(T_UD := JALOUSIE_UD_TIME_WINDOW_EG, T_ANGLE := t#1s);
wohnenJalousieS(T_UD := JALOUSIE_UD_TIME_WINDOW_EG, T_ANGLE:= t#1s);
wohnenJalousieWa(T_UD := JALOUSIE_UD_TIME_TERASSE, T_ANGLE:= t#1s);
wohnenJalousieWb(T_UD := JALOUSIE_UD_TIME_TERASSE, T_ANGLE:= t#1s);


(* output processing *)

kgGangLampe(ON := kgGangBwm.pulseOnMotion, PT := t#1m, ROOM := 'KG-Gang', LOCATION := 'Mitte');
kgEgLampe(ON_OFF := egGangTaster.pulseOnClick, PT := t#1m, ROOM := 'KG-EG-Stiege', LOCATION := 'Ost');
heizenLampe(ON_OFF := heizenTaster.pulseOnClick, PT := t#15m, ROOM := 'Heizen', LOCATION := 'West|Ost');
hobbyLampeS(ON := hobbyBwm.pulseOnMotion, ON_OFF := hobbyTasterR.pulseOnClick, PT := t#10m, ROOM := 'Hobby', LOCATION := 'Sued');
hobbyLampeN(ON := hobbyBwm.pulseOnMotion, ON_OFF := hobbyTasterL.pulseOnClick, PT := t#10m, ROOM := 'Hobby', LOCATION := 'Nord');
lagerLampe(ON := lagerBwm.pulseOnMotion, ON_OFF := lagerTasterNO.pulseOnClick, PT := t#3m, ROOM := 'Lager', LOCATION := 'Mitte');
lagerLampe.FORCE := vorratLampe.Q;
lagerLampe.FORCE_ON := vorratLampe.Q;
vorratLampe(ON_OFF := lagerTasterS.pulseOnClick, PT := t#2m, ROOM := 'Vorrat', LOCATION := 'Mitte');
waschenLampeNM(ON := waschenBwm.pulseOnMotion, ON_OFF := waschenTasterR.pulseOnClick, PT := t#15m, ROOM := 'Waschen', LOCATION := 'Nord|Mitte');
waschenLampeS(ON := waschenBwm.pulseOnMotion, ON_OFF := waschenTasterL.pulseOnClick, PT := t#15m, ROOM := 'Waschen', LOCATION := 'Sued');

egBadLampeON(
	ON_OFF := egBadTasterR.pulseOnLongpress
		OR egBadTasterL.pulseOnLongpress,
	PT := t#4h, ROOM := 'EG-Bad', LOCATION := 'Ost-Dusche');
egBadLampeOM(
	ON_OFF := egBadTasterL.pulseOnClick,
	PT := t#10m, ROOM := 'EG-Bad', LOCATION := 'Ost-Spiegel');
egBadLampeSM(
	ON_OFF := egBadTasterR.pulseOnClick,
	PT := t#30m, ROOM := 'EG-Bad', LOCATION := 'Sued|Mitte');
egBadDimmerSM(ON := egBadLampeSM.Q,
	INTENSITY := _dimmerEgBadSM_intensity,
	Status := _dimmerEgBadSM_status,
	DataIn := _dimmerEgBadSM_dataIn);
egGangLampe(ON := egGangBwm.pulseOnMotion,
	OFF := egGangTaster.pulseOnLongpress,
	OFF_BLOCK_ON := t#30s,
	PT := t#5m, ROOM := 'EG-Gang', LOCATION := 'Sued');
egWcLampe(
	ON := egWcBwm.pulseOnMotion,
	ON_OFF := egWcTaster.pulseOnClick,
	PT := t#6m, ROOM := 'EG-WC', LOCATION := 'West');
essenLampeM(
	ON_OFF := essenTasterO.pulseOnClick
		OR essenTasterR.pulseOnClick,
	PT := t#1h, ROOM := 'Essen', LOCATION := 'Mitte');
essenLampeS(
	ON_OFF := essenTasterO.pulseOnClick
		OR essenTasterL.pulseOnClick,
	PT := t#1h, ROOM := 'Essen', LOCATION := 'Sued');
essenLampeNW(
	ON_OFF := essenTasterO.pulseOnLongpress
		OR essenTasterR.pulseOnLongpress,
	PT := t#1h, ROOM := 'Essen', LOCATION := 'Sued');

kochenLampeO(
	ON_OFF := kochenTasterWO.pulseOnClick
		OR kochenTasterOR.pulseOnClick
		OR kochenTasterOL.pulseOnClick,
	ON := kochenBwm.pulseOnMotion,
	PT := t#1h, ROOM := 'Kochen', LOCATION := 'Ost');
kochenLampeN(
	ON_OFF := kochenTasterWR.pulseOnClick
		OR kochenTasterOL.pulseOnLongpress,
	PT := t#30m, ROOM := 'Kochen', LOCATION := 'Nord');
kochenLampeSW(
	ON_OFF := kochenTasterWL.pulseOnClick
		OR kochenTasterOR.pulseOnLongpress,
	PT := t#30m, ROOM := 'Kochen', LOCATION := 'Nord');

speisLampe(
	ON := speisTuer.pulseOnRelease,
	OFF := speisTuer.pulseOnPress,
	PT := t#5m, OFF_BLOCK_ON := T#0s, ROOM := 'Speis');

schlafenLampeS(
	ON_OFF := schlafenTasterOo.pulseOnClick
		OR schlafenTasterOr.pulseOnClick,
	OFF := schlafenTasterWML.pulseOnClick
		OR schlafenTasterWNR.pulseOnClick,
	PT := t#30m, ROOM := 'Schlafen', LOCATION := 'Sued');
schlafenLampeWM(ON_OFF := schlafenTasterWMR.pulseOnClick, PT := t#1h, ROOM := 'Schlafen', LOCATION := 'West-Mitte');
schlafenLampeWN(ON_OFF := schlafenTasterWNL.pulseOnClick, PT := t#1h, ROOM := 'Schlafen', LOCATION := 'West-Nord');
schlafenLampeO(
	ON_OFF := schlafenTasterOo.pulseOnClick
		OR schlafenTasterOl.pulseOnClick
		OR schlafenTasterWML.pulseOnClick
		OR schlafenTasterWNR.pulseOnClick,
	PT := t#30m, ROOM := 'Schlafen', LOCATION := 'Ost');
schlafenJalousieN();

wohnenLampeM(
	ON_OFF := wohnenTasterOO.pulseOnClick
		OR wohnenTasterWO.pulseOnClick,
	PT := t#1h, ROOM := 'Wohnen', LOCATION := 'Mitte');
wohnenLampeN(
	ON_OFF := wohnenTasterOL.pulseOnClick
		OR wohnenTasterWR.pulseOnClick,
	PT := t#1h, ROOM := 'Wohnen', LOCATION := 'Nord');
wohnenDimmerN(ON := wohnenLampeN.Q,
	INTENSITY := _dimmerWohnenN_intensity,
	Status := _dimmerWohnenN_status,
	DataIn := _dimmerWohnenN_dataIn);

wohnenLampeSW(
	ON_OFF := wohnenTasterOR.pulseOnClick
		OR wohnenTasterWL.pulseOnClick,
	PT := t#1h, ROOM := 'Wohnen', LOCATION := 'Sued-West');

egOgLampe(ON := ogGangBwm.pulseOnMotion,
	PT := t#5m, ROOM := 'EG-OG-Stiege', LOCATION := 'Ost');

arbeitenLampeN(
	ON_OFF := arbeitenTasterOO.pulseOnClick
		OR arbeitenTasterOL.pulseOnClick,
	PT := t#1h, ROOM := 'Arbeiten', LOCATION := 'Nord');
arbeitenLampeS(
	ON_OFF := arbeitenTasterOO.pulseOnClick
		OR arbeitenTasterOR.pulseOnClick,
	PT := t#1h, ROOM := 'Arbeiten', LOCATION := 'Sued');
arbeitenLampeSW(
	ON_OFF := arbeitenTasterOO.pulseOnLongpress
		OR arbeitenTasterOR.pulseOnLongpress,
	PT := t#1h, ROOM := 'Arbeiten', LOCATION := 'Sued-West');
ogBadLampeON(
	ON_OFF := ogBadTasterR.pulseOnLongpress
		OR ogBadTasterL.pulseOnLongpress,
	PT := t#10m, ROOM := 'OG-Bad', LOCATION := 'Ost-Dusche');
ogBadLampeOM(
	ON_OFF := ogBadTasterL.pulseOnClick,
	PT := t#10m, ROOM := 'OG-Bad', LOCATION := 'Ost-Spiegel');
ogBadLampeSM(
	ON_OFF := ogBadTasterR.pulseOnClick,
	PT := t#30m, ROOM := 'OG-Bad', LOCATION := 'Sued|Mitte');
ogGangLampe(ON := ogGangBwm.pulseOnMotion,
	PT := t#5m, ROOM := 'OG-Gang', LOCATION := 'Sued-West');
ogKindLampeM(
	ON_OFF := ogKindTasterNO.pulseOnClick,
	PT := t#1h, ROOM := 'OG-Kind', LOCATION := 'Mitte');
ogKindLampeN(
	ON_OFF := ogKindTasterNL.pulseOnClick,
	PT := t#1h, ROOM := 'OG-Kind', LOCATION := 'Nord');
ogKindLampeS(
	ON_OFF := ogKindTasterNR.pulseOnClick,
	PT := t#1h, ROOM := 'OG-Kind', LOCATION := 'Sued');
ogWcLampe(
	ON_OFF := ogWcTaster.pulseOnClick,
	PT := t#6m, ROOM := 'EG-WC', LOCATION := 'West');
gaesteLampeO(
	ON_OFF := gaesteTasterR.pulseOnClick
		OR gaesteTasterO.pulseOnClick,
	PT := t#1h, ROOM := 'Gaeste', LOCATION := 'Ost');
gaesteLampeW(
	ON_OFF := gaesteTasterL.pulseOnClick
		OR gaesteTasterO.pulseOnClick,
	PT := t#1h, ROOM := 'Gaeste', LOCATION := 'West');

dgKindLampe(ON_OFF := dgKindTaster.pulseOnClick,
	PT := t#2h, ROOM := 'DG-Kind', LOCATION := 'West-Sued');
dachbodenLampe(ON_OFF := dgKindTaster.pulseOnLongpress,
	PT := t#1h, ROOM := 'Dachboden', LOCATION := 'Ecke');

heizenHk1(soll := 24.0, vorlauf :=, ruecklauf :=);
heizenHk2(soll := 24.0, vorlauf :=, ruecklauf :=);

_lampeEgBadOM := egBadLampeOM.Q;
_lampeEgGang := egGangLampe.Q;
_lampeEgWc := egWcLampe.Q;
_lampeEssenM := essenLampeM.Q;
_lampeEssenS := essenLampeS.Q;
_lampeKochenSW := kochenLampeSW.Q;
_lampeOgGang := ogGangLampe.Q;
_lampeSchlafenS := schlafenLampeS.Q;
_lampeWohnenM := wohnenLampeM.Q;
_dimmerWohnenN_dataOut := wohnenDimmerN.DataOut;
_dimmerWohnenN_control := wohnenDimmerN.Control;
_dimmerEgBadSM_dataOut := egBadDimmerSM.DataOut;
_dimmerEgBadSM_control := egBadDimmerSM.Control;
END_PROGRAM

(* POU FBs/FB_Button, ST *)
FUNCTION_BLOCK FB_Button
VAR_INPUT
	ROOM: STRING;
	LOCATION: STRING;
	IN: BOOL;
	LONGPRESS: TIME := t#250ms; (*read by the visualisation*)
	RESET: BOOL := TRUE; (* if TRUE, viText is set; set to FALSE within the cycle *)
END_VAR
VAR_OUTPUT PERSISTENT
	toggleOnPress: BOOL;
	toggleOnRelease: BOOL;
	toggleOnLongpress: BOOL;
	toggleOnClick: BOOL;
	usageCounterPress: UDINT; (*overall number of press events*)
	usageCounterRelease: UDINT; (*overall number of release events*)
	usageCounterLongpress: UDINT; (*overall number longpress events*)
	usageCounterClick: UDINT; (*overall number of click events*)
END_VAR
VAR_OUTPUT
	isPressed: BOOL := FALSE;
	isReleased: BOOL; (*NOT isPressed*)
	isLongpressed: BOOL := FALSE;
	isClicked: BOOL := FALSE;
	pulseOnPress: BOOL;
	pulseOnRelease: BOOL;
	pulseOnLongpress: BOOL;
	pulseOnClick: BOOL; (* TAKE CARE: this is not reported after a pulseOnLongpress! if required, use pulseOnRelease. *)
END_VAR
VAR
	viIN: BOOL; (*written by the visualisation*)
	viText: STRING; (*read by the visualisation*)
	pTrig: R_TRIG;
	rTrig: F_TRIG;
	longpressTimer: TON;
	lTrig: R_TRIG;
	cTrig: R_TRIG;
	myIN: BOOL;
END_VAR
IF RESET THEN
	viText := CONCAT(ROOM, ' ');
	viText := CONCAT(viText, LOCATION);
	RESET := FALSE;
END_IF
myIN := IN XOR viIN;

pTrig(CLK := myIN);
rTrig(CLK := myIN);
pulseOnPress := pTrig.Q;
pulseOnRelease := rTrig.Q;

longpressTimer(IN := myIN, PT := LONGPRESS);
lTrig(CLK := longpressTimer.Q);
pulseOnLongpress := lTrig.Q;
IF pulseOnLongpress AND NOT pulseOnRelease THEN
	isLongpressed := TRUE;
	usageCounterLongpress := usageCounterLongpress + 1;
	toggleOnLongpress := fToggle(toggleOnLongpress);
ELSIF pulseOnLongpress THEN
	pulseOnLongpress := FALSE;
END_IF

IF pulseOnPress THEN
	isPressed := TRUE;
	isClicked := FALSE;
	isLongpressed := FALSE;
	usageCounterPress := usageCounterPress + 1;
	toggleOnPress := fToggle(toggleOnPress);
ELSIF pulseOnRelease THEN
	isPressed := FALSE;
	IF isLongpressed THEN
		isLongpressed := FALSE;
	ELSE
		isClicked := TRUE;
		usageCounterClick := usageCounterClick + 1;
		toggleOnClick := fToggle(toggleOnClick);
	END_IF
	usageCounterRelease := usageCounterRelease + 1;
	toggleOnRelease := fToggle(toggleOnRelease);
END_IF
isReleased := NOT isPressed;

cTrig(CLK := isClicked);
pulseOnClick := cTrig.Q;
END_FUNCTION_BLOCK

(* POU Fs/fToggle, ST *)
FUNCTION fToggle : BOOL
VAR_INPUT
	IN: BOOL;
END_VAR
IF IN THEN
	fToggle := FALSE;
ELSE
	fToggle := TRUE;
END_IF
END_FUNCTION

(* POU FBs/FB_Lamp, ST *)
(*
 TODO: REACTION
*)
FUNCTION_BLOCK FB_Lamp
VAR_INPUT
	ON_OFF: BOOL;   (* on/off on pulse, ignored if FORCE = TRUE *)
	ON: BOOL;   (* on on pulse, ignored if FORCE = TRUE *)
	OFF: BOOL;   (* off on pulse, ignored if FORCE = TRUE *)
	PT: TIME := t#30s;   (* auto-off aka on-time; see also: expandPT *)
	OFF_BLOCK_ON: TIME := t#15s;   (* after off block ON for the time specified *)
	REACTION: TIME := t#600ms;   (* TODO: do not change state right after statechange *)
	FORCE: BOOL;   (* if true, force output on/off, depending on FORCE_ON;
			  during FORCE, IN is ignored
			  during FORCE, PT is expanded if Q = TRUE *)
	FORCE_ON: BOOL;   (* if false and FORCE, then force off *)
	ROOM: STRING;
	LOCATION: STRING;
END_VAR
VAR_OUTPUT PERSISTENT
	usageTime: TIME := t#0ms;
	usageDays: UINT := 0;
	usageCounterSwitchOn: UDINT := 0;
END_VAR
VAR_OUTPUT
	Q: BOOL;   (* lamp on / off *)
END_VAR
VAR
	viText: STRING; (* ro by visualisation *)
	viOnTimer: TIME; (* ro by visualisation *)
	viOffTimer: TIME; (* ro by visualisation *)
	viOnOff: BOOL; (* wo by visualisation *)
	onTimer: TOF;
	offTimer: TOF;
	onTrigger: R_TRIG;
	onOffTrigger: R_TRIG;
	offTrigger: R_TRIG;
	forceOnTrigger: R_TRIG;
	forceOffTrigger: F_TRIG;
	forceOnTime: TIME;
	startOpTrigger: R_TRIG;
	stopOpTrigger: F_TRIG;
	opTimetracker: TIME;
	now: TIME;
	extendPT: TIME;   (* added to onTimer.PT *)
END_VAR
VAR CONSTANT
	MAX_TIME: TIME := T#71582m47s295ms;
END_VAR
viText := CONCAT(ROOM, '$N');
viText := CONCAT(viText, LOCATION);
(* viOnTimer and viOffTimer are set later *)

now := TIME();

forceOnTrigger(CLK := FORCE);
forceOffTrigger(CLK := FORCE);
IF forceOnTrigger.Q AND onTimer.Q THEN
	forceOnTime := now;
ELSIF forceOffTrigger.Q AND onTimer.Q THEN
	IF (now < forceOnTime) THEN
		(* overflow *)
		extendPT := MAX_TIME - forceOnTime + now;
	ELSE
		extendPT := now - forceOnTime;
	END_IF
	onTimer.PT := onTimer.PT + extendPT;
END_IF

IF FORCE THEN
	Q := FORCE_ON;
ELSE (* NOT FORCE *)
	onTrigger(CLK := ON);
	onOffTrigger(CLK := ON_OFF XOR viOnOff);
	offTrigger(CLK := OFF);
	IF (onTrigger.Q OR onOffTrigger.Q) AND NOT onTimer.Q THEN   (* on or on/off pulse and onTimer = off *)
		IF onTrigger.Q AND offTimer.Q THEN
			(* ignore on while offTimer.Q is TRUE *)
			;
		ELSE
			(* turn on lamp and onTimer, reset offTimer *)
			onTimer(IN := TRUE, PT := PT);
			offTimer(IN := FALSE, PT := OFF_BLOCK_ON);
		END_IF
	ELSIF (offTrigger.Q OR onOffTrigger.Q) AND onTimer.Q THEN   (* off or on/off pulse and onTimer = on *)
		(* turn off timer / lamp *)
		onTimer(IN := FALSE, PT := t#0s);
		extendPT := t#0ms;
		offTimer(IN := TRUE, PT := OFF_BLOCK_ON);
	ELSIF onTrigger.Q AND onTimer.Q THEN   (* on pulse and onTimer = on *)
		(* reset PT *)
		onTimer(IN := TRUE, PT := PT);
 	ELSIF onTimer.Q THEN   (* no on/off pulse but timer is on *)
		onTimer(IN := FALSE);
	ELSIF offTimer.Q THEN
		offTimer(IN := FALSE);
	END_IF
	Q := onTimer.Q;
END_IF (* NOT FORCE *)

IF onTimer.ET = onTimer.PT THEN
	(* we do not want to see 0, when the onTimer is finished *)
	(* instead, display PT *)
	viOnTimer := PT;
ELSE
	viOnTimer := onTimer.PT - onTimer.ET;
END_IF
IF offTimer.ET = offTimer.PT THEN
	(* we do not want to see 0, when the offTimer is finished *)
	(* instead, display PT *)
	viOffTimer := OFF_BLOCK_ON;
ELSE
	viOffTimer := offTimer.PT - offTimer.ET;
END_IF

(*****************************)
(* record the operation time *)

startOpTrigger(CLK := Q);
stopOpTrigger(CLK := Q);
IF startOpTrigger.Q THEN
	usageCounterSwitchOn := usageCounterSwitchOn + 1;
	opTimetracker := now;
END_IF
IF Q AND (now < opTimetracker) THEN   (* overflow *)
	usageTime := usageTime + (MAX_TIME - opTimetracker);
	opTimetracker := t#0ms;
END_IF
IF stopOpTrigger.Q THEN
	usageTime := usageTime + (now - opTimetracker);
END_IF
IF Q AND ((now - opTimetracker) > t#1s) THEN
	usageTime := usageTime + (now - opTimetracker);
	opTimetracker := now;
END_IF
IF (Q OR stopOpTrigger.Q) AND (usageTime > t#1d) THEN
	usageDays := usageDays + 1;
	usageTime := usageTime - t#1d;
END_IF
END_FUNCTION_BLOCK

(* POU FBs/FB_Heizkreis, ST *)
FUNCTION_BLOCK FB_Heizkreis
VAR_INPUT
	soll:REAL;
	vorlauf: REAL;
	ruecklauf: REAL;
END_VAR
VAR_OUTPUT
	mischer AT %Q*: INT;   (* 0x7FFF = 100% = 10V; 0x0000 = 0% = 0V*)
	pumpe AT %Q*: INT;   (* 0x7FFF = 100% = 10V; 0x0000 = 0% = 0V*)
END_VAR
VAR
END_VAR
mischer := 6000;
pumpe := 0;
END_FUNCTION_BLOCK

(* POU FBs/FB_Motion, ST *)
FUNCTION_BLOCK FB_Motion
VAR_INPUT
	IN: BOOL;
	ROOM: STRING;
	LOCATION: STRING;
END_VAR
VAR_OUTPUT
	Q: BOOL;
	pulseOnMotion: BOOL;
END_VAR
VAR
	viText: STRING;
	viIN: BOOL;
	myIN: BOOL;
	x: R_TRIG;
END_VAR
(* support VIsualisations *)
viText := CONCAT(ROOM, '$N');
viText := CONCAT(viText, LOCATION);
myIN := IN XOR viIN;

Q := myIN;
x(CLK := myIn);
pulseOnMotion := x.Q;
END_FUNCTION_BLOCK

(* POU FBs/FB_Light, ST *)
FUNCTION_BLOCK FB_Light
VAR_INPUT
	Status: USINT;
	DataIn: INT;
	ROOM: STRING;
	LOCATION: STRING;
END_VAR
VAR_OUTPUT
	Value: REAL;
	Error: BOOL;
END_VAR
VAR
	viText: STRING;
END_VAR
(* support VIsualisations *)
viText := CONCAT(ROOM, '$N');
viText := CONCAT(viText, LOCATION);

Error := TRUE;
Value := INT_TO_REAL(DataIn);
END_FUNCTION_BLOCK

(* POU FBs/FB_Temperature, ST *)
FUNCTION_BLOCK FB_Temperature
VAR_INPUT
	Status: USINT;
	DataIn: INT;
	UNIT: E_TemperatureUnit;
	ROOM: STRING;
	LOCATION: STRING;
END_VAR
VAR_OUTPUT
	Value: REAL;
	Error: BOOL;
END_VAR
VAR
	viText: STRING;
END_VAR
(* support VIsualisations *)
viText := CONCAT(ROOM, '$N');
viText := CONCAT(viText, LOCATION);

IF Status.6 THEN
	Error := TRUE;
ELSE
	Error := FALSE;
	Value := INT_TO_REAL(DataIn) / 100;
END_IF
END_FUNCTION_BLOCK

(* POU FBs/FB_Dimmer, ST *)
FUNCTION_BLOCK FB_Dimmer
VAR_INPUT
	ON: BOOL;
	INTENSITY: REAL; (* 0..100; clamped *)
	Status: USINT;
	DataIn: INT;
END_VAR
VAR_OUTPUT
	Control: USINT;
	DataOut: INT;
END_VAR
VAR
	mIntensity: REAL;
	mLastIntensity: REAL;
END_VAR
(*
KL2751: 300VA (1.35A)
KL2761: 600VA (2.7A)

wo: DataOut: 0..32767
wo: Control.7: 1=registerAccess, 0=processData
wo: Control.6: if Control.7=1: 0=readRegister, 1=writeRegister
wo: Control.5-0: if Control.7=1: register
wo: Control.0: if Control.7=0: manual autodetect (0->1) 
ro: DataIn: Internal temperature in celsius
ro: Status.7: 1=registerAccess, 0=processData
if Status.7=0=processData:
ro: Status.6: error (short)
ro: Status.5: temperature warning (>80 grad celsius) - 20% max til 60 grad celsius
ro: Status.4: overload (on turn on)
ro: Status.3: operation mode 0=auto 1=abschnitt 2=anschnitt
ro: Status.2: operation mode 3=posHalbwelleAnschnitt
ro: Status.1: operation mode 4=negHalbwelleAnschnitt
ro: Status.0: synchron
if Status.7=1=registerAccess:
ro: Status.6: 0=readRegister, 1=writeRegister
ro: Status.5-0: register

rw  r7    (ram): command
ro  r8    (rom): hw type: 2751 or 2761 (dec) = "2751" or "2761"
ro  r9    (rom): fw version: 0x3141 = "1A"
ro r10    (rom): multiplex shift
ro r11    (rom): signal channels
ro r12    (rom): min datalength
ro r13    (rom): data structure
rw r15    (ram): alignment
rw r16 (eeprom): hw version
ro r29    (rom): hw subtype: 0x000b = 11 = "-0011"
rw r31    (ram): codeword 0x1235=rwOtherRegister def(<>0x1235)=roOtherRegister
rw r32 (eeprom): feature
   r32.3: dimRamp 0(def)=rel 1=abs(anyChangeUsesFullTime)
   r32.2: disWatchdog
   r32.0: enUserScale (r33/r34)
rw r33 (eeprom): scale-offset
rw r34 (eeprom): scale-gain 0x100(def)=1 0x80=0.5 0x200=2 ...
rw r35 (eeprom): ramp time 0=50ms 1=100ms 2=200ms 3(def)=500ms 4=1s 5=2s 6=5s 7=10s
rw r36 (eeprom): watchdog-timeout 10(dec)=100ms 22(dec)=220ms ...
rw r37 (eeprom): timeout (k-bus error) on-value def=16383(dec)
rw r38 (eeprom): timeout (k-bus error) off-value def=0
rw r39 (eeprom): dimmer mode (see Status.3-1)
rw r40 (eeprom): after short 0=stayOff 1(def)=turnOn
rw r41 (eeprom): frequency 0(def)=50hz 1=60hz

r7 command 0x7000: factory reset

I. Schreiben des Code-Worts (0x1235) in Register 31
II. Lesen des Register 31 (gesetztes Code-Wort überprüfen)
III. Schreiben des Register 32 (Inhalt des Feature-Registers ändern)
IV. Lesen des Register 32 (geändertes Feature-Register überprüfen)
V. Schreiben des Register 31 (Code-Wort zurücksetzen)

*)

IF NOT ON OR INTENSITY < 0 THEN
	mIntensity := 0;
ELSIF INTENSITY > 100 THEN
	mIntensity := 100;
ELSE
	mIntensity := INTENSITY;
END_IF

IF mIntensity <> mLastIntensity THEN
	Control := 0;
	DataOut := REAL_TO_INT(mIntensity * 16#7FFF / 100);
	mLastIntensity := mIntensity;
END_IF
END_FUNCTION_BLOCK

(* POU FBs/FB_Jalousie, ST *)
FUNCTION_BLOCK FB_Jalousie
VAR_INPUT
	T_UD: TIME;
	T_ANGLE: TIME;
	PI: BYTE;
	AI: BYTE;
	UD: TIME := t#10s;
	ANGLE: TIME := t#3s;
END_VAR
VAR_OUTPUT
	Qu AT %Q*: BOOL;
	Qd AT %Q*: BOOL;
END_VAR
VAR
	viUp: BOOL;
	viDown: BOOL;
	viAuto: BOOL;
	mInput: BLIND_INPUT;
	(* mActuator: BLIND_ACTUATOR;  integrated in BLIND_CONTROL *)
	mControl: BLIND_CONTROL;
END_VAR
(* mControl.SENS := 0; *)
mControl.T_UD := T_UD;
mControl.T_ANGLE := T_ANGLE;

mControl.PI := PI;

mInput(S1 := viUp, S2 := viDown, IN := viAuto, POS := mControl.POS, ANG := mControl.ANG);
mControl(UP := mInput.QU, DN := mInput.QD, S_IN := mInput.STATUS, PI := mInput.PO, AI := mInput.AO);

Qu := mControl.MU;
Qd := mControl.MD;
END_FUNCTION_BLOCK

(* POU MAIN_SLOW, ST *)
PROGRAM MAIN_SLOW
VAR_OUTPUT

END_VAR
VAR
	fbDoubleButton: FB_DoubleButton;
END_VAR
fbDoubleButton(CLICK_A_IN := MAIN.schlafenTasterOl.isClicked, CLICK_B_IN := MAIN.schlafenTasterOr.isClicked);
END_PROGRAM

(* POU FBs/FB_DoubleButton, ST *)
FUNCTION_BLOCK FB_DoubleButton
VAR_INPUT
	ACTIVITY: BOOL;
	RESET: BOOL := TRUE;
	FALLBACK: TIME := t#15s;
	TIMEOUT: TIME := t#250ms;
	CLICK_A_IN: BOOL;
	CLICK_B_IN: BOOL;
	LONGCLICK_A_IN: BOOL;
	LONGCLICK_B_IN: BOOL;
END_VAR
VAR_OUTPUT
	Q: UINT; (* counts the doublepresses, resets to 0 after FALLBACK *)
	CLICK_A_OUT: BOOL;
	CLICK_B_OUT: BOOL;
	LONGCLICK_A_OUT: BOOL;
	LONGCLICK_B_OUT: BOOL;
END_VAR
VAR
	rA: R_TRIG;
	rB: R_TRIG;
	lTof: TOF;
	rTof: TOF;
	timer: TON;
	manual: BOOL;
	reStart: R_TRIG;
END_VAR
IF RESET THEN
	Q := 0;
	timer(IN := FALSE); (* reset timer *)
	RESET := FALSE;
END_IF

IF Q > 0 THEN
	IF ACTIVITY THEN (* advance timer *)
		timer(IN := FALSE);
		timer.IN := TRUE;
	END_IF
	timer(); (* update timer *)
	IF timer.Q = TRUE THEN
		RESET := TRUE;
	END_IF
END_IF

rA(CLK := CLICK_A_IN);
rB(CLK := CLICK_B_IN);
lTof(IN := rA.Q, PT := TIMEOUT);
rTof(IN := rB.Q, PT := TIMEOUT);
reStart(CLK := lTof.Q AND rTof.Q);

IF reStart.Q THEN
	Q := Q + 1;
	IF Q = 1 THEN (* init timer *)
		timer.IN := TRUE;
		timer.PT := FALLBACK;
	ELSE
		timer(IN := FALSE);
		timer.IN := TRUE;
	END_IF
	timer(); (* update timer *)
END_IF
END_FUNCTION_BLOCK

(* POU MAIN_FAST, ST *)
PROGRAM MAIN_FAST
VAR CONSTANT
	FROELING_MODBUS_ADDRESS: USINT := 9;
END_VAR
VAR
	rs232: FB_SetSerial;
	fbFroeling: FB_Froeling;
(*	froeling: ModbusRtuMaster_KL6x22B;
	froelingIn: MB_KL6inData22B;
	froelingOut: MB_KL6outData22B;
	froelingData: INT;
*)
	uiStateCX5000 AT %I*: UINT;
	uiControlCX5000 AT %Q* : UINT;
	iVoltagePhase1 AT %I* : ARRAY [0..9] OF INT;
	iVoltagePhase2 AT %I* : ARRAY [0..9] OF INT;
	iVoltagePhase3 AT %I* : ARRAY [0..9] OF INT;
	uliStartTimeNextLatch AT %I* : ARRAY [0..1] OF UDINT;
	bWcState AT %I* : BOOL;

	fbAnalyseVoltagePhase1 : FB_ANALYSE_VOLTAGE;
	fbAnalyseVoltagePhase2 : FB_ANALYSE_VOLTAGE;
	fbAnalyseVoltagePhase3 : FB_ANALYSE_VOLTAGE;
	fbA28CH1: FB_SYNC_RELAIS;
	fbA28CH2: FB_SYNC_RELAIS;
	fbA29CH1: FB_SYNC_RELAIS;
	fbA29CH2: FB_SYNC_RELAIS;
	fbA30CH1: FB_SYNC_RELAIS;
	fbA30CH2: FB_SYNC_RELAIS;
	fbA31CH1: FB_SYNC_RELAIS;
	fbA31CH2: FB_SYNC_RELAIS;
	fbA32CH1: FB_SYNC_RELAIS;
	fbA32CH2: FB_SYNC_RELAIS;
	fbA20CH1: FB_SYNC_RELAIS;
	fbA20CH2: FB_SYNC_RELAIS;
	fbA21CH1: FB_SYNC_RELAIS;
	fbA21CH2: FB_SYNC_RELAIS;
	fbA23CH1: FB_SYNC_RELAIS;
	fbA23CH2: FB_SYNC_RELAIS;
	fbA24CH1: FB_SYNC_RELAIS;
	fbA24CH2: FB_SYNC_RELAIS;
	fbA25CH1: FB_SYNC_RELAIS;
	fbA25CH2: FB_SYNC_RELAIS;
	fbA26CH1: FB_SYNC_RELAIS;
	fbA26CH2: FB_SYNC_RELAIS;
	fbA38OGCH1: FB_SYNC_RELAIS;
	fbA38OGCH2: FB_SYNC_RELAIS;
	fbA41OGCH1: FB_SYNC_RELAIS;
	fbA41OGCH2: FB_SYNC_RELAIS;
	fbA43OGCH1: FB_SYNC_RELAIS;
	fbA43OGCH2: FB_SYNC_RELAIS;
	fbA44OGCH1: FB_SYNC_RELAIS;
	fbA44OGCH2: FB_SYNC_RELAIS;
	fbA45OGCH1: FB_SYNC_RELAIS;
	fbA45OGCH2: FB_SYNC_RELAIS;
	fbA48OGCH1: FB_SYNC_RELAIS;
	fbA48OGCH2: FB_SYNC_RELAIS;
	fbA49OGCH1: FB_SYNC_RELAIS;
	fbA49OGCH2: FB_SYNC_RELAIS;
	fbA50OGCH1: FB_SYNC_RELAIS;
	fbA50OGCH2: FB_SYNC_RELAIS;
	fbA52OGCH1: FB_SYNC_RELAIS;
	fbA52OGCH2: FB_SYNC_RELAIS;
	fbA53OGCH1: FB_SYNC_RELAIS;
	fbA53OGCH2: FB_SYNC_RELAIS;
	fbA55OGCH1: FB_SYNC_RELAIS;
	fbA55OGCH2: FB_SYNC_RELAIS;
	fbA56OGCH1: FB_SYNC_RELAIS;
	fbA56OGCH2: FB_SYNC_RELAIS;
	fbA57OGCH1: FB_SYNC_RELAIS;
	fbA57OGCH2: FB_SYNC_RELAIS;
	fbA15OGCH1: FB_SYNC_RELAIS;
	fbA15OGCH2: FB_SYNC_RELAIS;
	fbA17OGCH1: FB_SYNC_RELAIS;
	fbA17OGCH2: FB_SYNC_RELAIS;
	fbA18OGCH1: FB_SYNC_RELAIS;
	fbA18OGCH2: FB_SYNC_RELAIS;
	fbA19OGCH1: FB_SYNC_RELAIS;
	fbA19OGCH2: FB_SYNC_RELAIS;
	fbA21OGCH1: FB_SYNC_RELAIS;
	fbA21OGCH2: FB_SYNC_RELAIS;
	fbA23OGCH1: FB_SYNC_RELAIS;
	fbA23OGCH2: FB_SYNC_RELAIS;
	fbA25OGCH1: FB_SYNC_RELAIS;
	fbA25OGCH2: FB_SYNC_RELAIS;
	fbA26OGCH1: FB_SYNC_RELAIS;
	fbA26OGCH2: FB_SYNC_RELAIS;
	fbA33OGCH1: FB_SYNC_RELAIS;
	fbA33OGCH2: FB_SYNC_RELAIS;
	fbA35OGCH1: FB_SYNC_RELAIS;
	fbA35OGCH2: FB_SYNC_RELAIS;
	fbA36OGCH1: FB_SYNC_RELAIS;
	fbA36OGCH2: FB_SYNC_RELAIS;
	fbA78OGCH1: FB_SYNC_RELAIS;
	fbA78OGCH2: FB_SYNC_RELAIS;
	fbA80OGCH1: FB_SYNC_RELAIS;
	fbA80OGCH2: FB_SYNC_RELAIS;

	lrFrequencyPhase1: LREAL;
	lrFrequencyPhase2: LREAL;
	lrFrequencyPhase3: LREAL;
	bErrorL1: BOOL;
	bErrorL2: BOOL;
	bErrorL3: BOOL;

	bRelayPLC:BOOL;
END_VAR
(*
froeling.UnitID := 10;
froeling.Quantity := 1;
froeling.MBAddr := 30022;
froeling.cbLength := SIZEOF(froelingData);
froeling.pMemoryAddr := ADR(froelingData);
froeling.Timeout := t#8s;
froeling.Execute := TRUE;
*)

fbFroeling(
	modbusSlaveAddress := FROELING_MODBUS_ADDRESS,
	timeout := t#1s,
);

(* Spannungsanalyse *)
fbAnalyseVoltagePhase1(
	uliStartTimeNextLatch := uliStartTimeNextLatch,
	bWcState := bWcState,
	iVoltage := iVoltagePhase1,
	lrFrequency => lrFrequencyPhase1,
	bError => bErrorL1);

fbAnalyseVoltagePhase2(
	uliStartTimeNextLatch := uliStartTimeNextLatch,
	bWcState := bWcState,
	iVoltage := iVoltagePhase2,
	lrFrequency => lrFrequencyPhase2,
	bError => bErrorL2);

fbAnalyseVoltagePhase3(
	uliStartTimeNextLatch := uliStartTimeNextLatch,
	bWcState := bWcState,
	iVoltage := iVoltagePhase3,
	lrFrequency => lrFrequencyPhase3,
	bError => bErrorL3);

(* Relais *)
fbA28CH1(bValue:= , udiDelayNanoSek:= 5800000, tNextZeroVoltage:= fbAnalyseVoltagePhase1.tNextZeroVoltage);
fbA28CH2(bValue:= , udiDelayNanoSek:= 6600000, tNextZeroVoltage:= fbAnalyseVoltagePhase1.tNextZeroVoltage);
fbA29CH1(bValue:= , udiDelayNanoSek:= 6300000, tNextZeroVoltage:= fbAnalyseVoltagePhase1.tNextZeroVoltage);
fbA29CH2(bValue:= , udiDelayNanoSek:= 6500000, tNextZeroVoltage:= fbAnalyseVoltagePhase1.tNextZeroVoltage);
fbA30CH1(bValue:= , udiDelayNanoSek:= 6500000, tNextZeroVoltage:= fbAnalyseVoltagePhase1.tNextZeroVoltage);
fbA30CH2(bValue:= , udiDelayNanoSek:= 5700000, tNextZeroVoltage:= fbAnalyseVoltagePhase1.tNextZeroVoltage);
fbA31CH1(bValue:= , udiDelayNanoSek:= 5700000, tNextZeroVoltage:= fbAnalyseVoltagePhase1.tNextZeroVoltage);
fbA31CH2(bValue:= , udiDelayNanoSek:= 5700000, tNextZeroVoltage:= fbAnalyseVoltagePhase1.tNextZeroVoltage);
fbA32CH1(bValue:= , udiDelayNanoSek:= 6000000, tNextZeroVoltage:= fbAnalyseVoltagePhase2.tNextZeroVoltage);
fbA32CH2(bValue:= , udiDelayNanoSek:= 6000000, tNextZeroVoltage:= fbAnalyseVoltagePhase2.tNextZeroVoltage);
fbA20CH1(bValue:=MAIN.kgGangLampe.Q, udiDelayNanoSek:= 6700000, tNextZeroVoltage:= fbAnalyseVoltagePhase1.tNextZeroVoltage);
fbA20CH2(bValue:=MAIN.kgEgLampe.Q, udiDelayNanoSek:= 5800000, tNextZeroVoltage:= fbAnalyseVoltagePhase1.tNextZeroVoltage);
fbA21CH1(bValue:=MAIN.lagerLampe.Q, udiDelayNanoSek:= 6400000, tNextZeroVoltage:= fbAnalyseVoltagePhase1.tNextZeroVoltage);
fbA21CH2(bValue:= , udiDelayNanoSek:= 6500000, tNextZeroVoltage:= fbAnalyseVoltagePhase1.tNextZeroVoltage);
fbA23CH1(bValue:=MAIN.heizenLampe.Q, udiDelayNanoSek:= 6500000, tNextZeroVoltage:= fbAnalyseVoltagePhase2.tNextZeroVoltage);
fbA23CH2(bValue:=MAIN.waschenLampeS.Q, udiDelayNanoSek:= 6300000, tNextZeroVoltage:= fbAnalyseVoltagePhase2.tNextZeroVoltage);
fbA24CH1(bValue:=MAIN.waschenLampeNM.Q, udiDelayNanoSek:= 6300000, tNextZeroVoltage:= fbAnalyseVoltagePhase2.tNextZeroVoltage);
fbA24CH2(bValue:=MAIN.hobbyLampeN.Q, udiDelayNanoSek:= 6000000, tNextZeroVoltage:= fbAnalyseVoltagePhase2.tNextZeroVoltage);
fbA25CH1(bValue:=MAIN.vorratLampe.Q, udiDelayNanoSek:= 6000000, tNextZeroVoltage:= fbAnalyseVoltagePhase2.tNextZeroVoltage);
fbA25CH2(bValue:=MAIN.hobbyLampeS.Q, udiDelayNanoSek:= 6300000, tNextZeroVoltage:= fbAnalyseVoltagePhase2.tNextZeroVoltage);
fbA26CH1(bValue:= , udiDelayNanoSek:= 6300000, tNextZeroVoltage:= fbAnalyseVoltagePhase2.tNextZeroVoltage);
fbA26CH2(bValue:= , udiDelayNanoSek:= 6150000, tNextZeroVoltage:= fbAnalyseVoltagePhase2.tNextZeroVoltage);
fbA38OGCH1(bValue:= , udiDelayNanoSek:= 6000000, tNextZeroVoltage:= fbAnalyseVoltagePhase1.tNextZeroVoltage);
fbA38OGCH2(bValue:= , udiDelayNanoSek:= 6200000, tNextZeroVoltage:= fbAnalyseVoltagePhase1.tNextZeroVoltage);
fbA41OGCH1(bValue:= , udiDelayNanoSek:= 6200000, tNextZeroVoltage:= fbAnalyseVoltagePhase2.tNextZeroVoltage);
fbA41OGCH2(bValue:=MAIN.ogBadLampeOM.Q, udiDelayNanoSek:= 5600000, tNextZeroVoltage:= fbAnalyseVoltagePhase2.tNextZeroVoltage);
fbA43OGCH1(bValue:= , udiDelayNanoSek:= 5800000, tNextZeroVoltage:= fbAnalyseVoltagePhase1.tNextZeroVoltage);
fbA43OGCH2(bValue:= , udiDelayNanoSek:= 5800000, tNextZeroVoltage:= fbAnalyseVoltagePhase1.tNextZeroVoltage);
fbA44OGCH1(bValue:=MAIN.ogKindLampeN.Q, udiDelayNanoSek:= 5800000, tNextZeroVoltage:= fbAnalyseVoltagePhase1.tNextZeroVoltage);
fbA44OGCH2(bValue:=MAIN.ogKindLampeS.Q, udiDelayNanoSek:= 5800000, tNextZeroVoltage:= fbAnalyseVoltagePhase1.tNextZeroVoltage);
fbA45OGCH1(bValue:=MAIN.ogKindLampeM.Q, udiDelayNanoSek:= 5800000, tNextZeroVoltage:= fbAnalyseVoltagePhase1.tNextZeroVoltage);
fbA45OGCH2(bValue:=MAIN.dgKindLampe.Q, udiDelayNanoSek:= 5800000, tNextZeroVoltage:= fbAnalyseVoltagePhase1.tNextZeroVoltage);
fbA48OGCH1(bValue:= , udiDelayNanoSek:= 6000000, tNextZeroVoltage:= fbAnalyseVoltagePhase2.tNextZeroVoltage);
fbA48OGCH2(bValue:= , udiDelayNanoSek:= 6000000, tNextZeroVoltage:= fbAnalyseVoltagePhase2.tNextZeroVoltage);
fbA49OGCH1(bValue:= , udiDelayNanoSek:= 6000000, tNextZeroVoltage:= fbAnalyseVoltagePhase2.tNextZeroVoltage);
fbA49OGCH2(bValue:= , udiDelayNanoSek:= 5800000, tNextZeroVoltage:= fbAnalyseVoltagePhase2.tNextZeroVoltage);
fbA50OGCH1(bValue:= , udiDelayNanoSek:= 6000000, tNextZeroVoltage:= fbAnalyseVoltagePhase2.tNextZeroVoltage);
fbA50OGCH2(bValue:= , udiDelayNanoSek:= 5600000, tNextZeroVoltage:= fbAnalyseVoltagePhase2.tNextZeroVoltage);
fbA52OGCH1(bValue:= , udiDelayNanoSek:= 6000000, tNextZeroVoltage:= fbAnalyseVoltagePhase2.tNextZeroVoltage);
fbA52OGCH2(bValue:= , udiDelayNanoSek:= 6000000, tNextZeroVoltage:= fbAnalyseVoltagePhase2.tNextZeroVoltage);
fbA53OGCH1(bValue:= , udiDelayNanoSek:= 5900000, tNextZeroVoltage:= fbAnalyseVoltagePhase2.tNextZeroVoltage);
fbA53OGCH2(bValue:= , udiDelayNanoSek:= 5900000, tNextZeroVoltage:= fbAnalyseVoltagePhase2.tNextZeroVoltage);
fbA55OGCH1(bValue:= , udiDelayNanoSek:= 5900000, tNextZeroVoltage:= fbAnalyseVoltagePhase3.tNextZeroVoltage);
fbA55OGCH2(bValue:= , udiDelayNanoSek:= 5600000, tNextZeroVoltage:= fbAnalyseVoltagePhase3.tNextZeroVoltage);
fbA56OGCH1(bValue:= , udiDelayNanoSek:= 5600000, tNextZeroVoltage:= fbAnalyseVoltagePhase3.tNextZeroVoltage);
fbA56OGCH2(bValue:= , udiDelayNanoSek:= 5700000, tNextZeroVoltage:= fbAnalyseVoltagePhase3.tNextZeroVoltage);
fbA57OGCH1(bValue:= , udiDelayNanoSek:= 5600000, tNextZeroVoltage:= fbAnalyseVoltagePhase3.tNextZeroVoltage);
fbA57OGCH2(bValue:= , udiDelayNanoSek:= 5900000, tNextZeroVoltage:= fbAnalyseVoltagePhase3.tNextZeroVoltage);

fbA15OGCH1(bValue:=MAIN.essenLampeNW.Q, udiDelayNanoSek:= 6100000, tNextZeroVoltage:= fbAnalyseVoltagePhase1.tNextZeroVoltage);
fbA15OGCH2(bValue:= , udiDelayNanoSek:= 6300000, tNextZeroVoltage:= fbAnalyseVoltagePhase1.tNextZeroVoltage);
fbA17OGCH1(bValue:=MAIN.schlafenLampeO.Q, udiDelayNanoSek:= 6100000, tNextZeroVoltage:= fbAnalyseVoltagePhase2.tNextZeroVoltage);
fbA17OGCH2(bValue:= , udiDelayNanoSek:= 6100000, tNextZeroVoltage:= fbAnalyseVoltagePhase2.tNextZeroVoltage);
fbA18OGCH1(bValue:=MAIN.wohnenLampeSW.Q, udiDelayNanoSek:= 6100000, tNextZeroVoltage:= fbAnalyseVoltagePhase2.tNextZeroVoltage);
fbA18OGCH2(bValue:= , udiDelayNanoSek:= 6100000, tNextZeroVoltage:= fbAnalyseVoltagePhase2.tNextZeroVoltage);
fbA19OGCH1(bValue:= , udiDelayNanoSek:= 6100000, tNextZeroVoltage:= fbAnalyseVoltagePhase2.tNextZeroVoltage);
fbA19OGCH2(bValue:= , udiDelayNanoSek:= 6100000, tNextZeroVoltage:= fbAnalyseVoltagePhase2.tNextZeroVoltage);
fbA21OGCH1(bValue:= , udiDelayNanoSek:= 6000000, tNextZeroVoltage:= fbAnalyseVoltagePhase3.tNextZeroVoltage);
fbA21OGCH2(bValue:= , udiDelayNanoSek:= 6100000, tNextZeroVoltage:= fbAnalyseVoltagePhase3.tNextZeroVoltage);
fbA23OGCH1(bValue:= , udiDelayNanoSek:= 6100000, tNextZeroVoltage:= fbAnalyseVoltagePhase2.tNextZeroVoltage);
fbA23OGCH2(bValue:= , udiDelayNanoSek:= 6100000, tNextZeroVoltage:= fbAnalyseVoltagePhase2.tNextZeroVoltage);
fbA25OGCH1(bValue:=MAIN.kochenLampeO.Q, udiDelayNanoSek:= 6100000, tNextZeroVoltage:= fbAnalyseVoltagePhase2.tNextZeroVoltage);
fbA25OGCH2(bValue:=MAIN.kochenLampeN.Q, udiDelayNanoSek:= 6100000, tNextZeroVoltage:= fbAnalyseVoltagePhase2.tNextZeroVoltage);
fbA26OGCH1(bValue:=MAIN.speisLampe.Q , udiDelayNanoSek:= 6100000, tNextZeroVoltage:= fbAnalyseVoltagePhase2.tNextZeroVoltage);
fbA26OGCH2(bValue:= , udiDelayNanoSek:= 6100000, tNextZeroVoltage:= fbAnalyseVoltagePhase2.tNextZeroVoltage);
fbA33OGCH1(bValue:=MAIN.egBadLampeON.Q, udiDelayNanoSek:= 6100000, tNextZeroVoltage:= fbAnalyseVoltagePhase1.tNextZeroVoltage);
fbA33OGCH2(bValue:= , udiDelayNanoSek:= 6100000, tNextZeroVoltage:= fbAnalyseVoltagePhase1.tNextZeroVoltage);
fbA35OGCH1(bValue:=MAIN.arbeitenLampeN.Q, udiDelayNanoSek:= 6300000, tNextZeroVoltage:= fbAnalyseVoltagePhase3.tNextZeroVoltage);
fbA35OGCH2(bValue:=MAIN.arbeitenLampeS.Q, udiDelayNanoSek:= 6200000, tNextZeroVoltage:= fbAnalyseVoltagePhase3.tNextZeroVoltage);
fbA36OGCH1(bValue:=MAIN.arbeitenLampeSW.Q, udiDelayNanoSek:= 6400000, tNextZeroVoltage:= fbAnalyseVoltagePhase3.tNextZeroVoltage);
fbA36OGCH2(bValue:= , udiDelayNanoSek:= 6300000, tNextZeroVoltage:= fbAnalyseVoltagePhase3.tNextZeroVoltage);
fbA78OGCH1(bValue:= , udiDelayNanoSek:= 5800000, tNextZeroVoltage:= fbAnalyseVoltagePhase3.tNextZeroVoltage);
fbA78OGCH2(bValue:=MAIN.dachbodenLampe.Q, udiDelayNanoSek:= 5800000, tNextZeroVoltage:= fbAnalyseVoltagePhase3.tNextZeroVoltage);
fbA80OGCH1(bValue:= , udiDelayNanoSek:= 5500000, tNextZeroVoltage:= fbAnalyseVoltagePhase1.tNextZeroVoltage);
fbA80OGCH2(bValue:= , udiDelayNanoSek:= 5500000, tNextZeroVoltage:= fbAnalyseVoltagePhase1.tNextZeroVoltage);
END_PROGRAM

(* POU FBs/FB_SetSerial, ST *)
(*
	EL6001 / EL6021:
		864 bytes receive buffer
		128 bytes transmit buffer
		2400 … 115200 baud
		default: 9600 baud, 8 data bits, no parity, one stop bit
		22 x 8 bit input, 22 x 8 bit output, 16 bit control, 16 bit status
		1008:0 Device name STRING RO "EL6001" "EL6021"
		1009:0 Hardware version STRING RO "04"
		100A:0 Software version STRING RO "05"
		4073:0 Baudrate  UINT16 RW 0x0006
		4074:0 Dataframe UINT16 RW 0x0003
		4075:01 0: RTS/CTS disabled | Full duplex mode 
		        1: RTS/CTS  enabled | Half duplex mode BOOLEAN RW 0x00
		4075:02 0: TX XON/XOFF not supported
		        1: TX XON/XOFF     supported BOOLEAN RW 0x00
		4075:03 0: RX XON/XOFF not supported
		        1: RX XON/XOFF     supported BOOLEAN RW 0x00
*)
FUNCTION_BLOCK FB_SetSerial
VAR_INPUT
	BAUDRATE: Baudrate := B9600;
	RTS_CTS: BOOL := FALSE;
	RX_XON_XOFF: BOOL := FALSE;
	TX_XON_XOFF: BOOL := FALSE;
	EXECUTE: BOOL := FALSE;
END_VAR
VAR_OUTPUT
	busy: BOOL;
END_VAR
VAR
	execTrigger: R_TRIG;
	fbSdoRead 	: FB_EcCoESdoRead;
(*
	TYPE T_AmsNetId : STRING(23);
	END_TYPE
	Eine SPS-Variable von diesem Typ ist ein STRING, der
	die AMS-Netzwerkkennung des Zielgerätes enthäLT, an
	das der ADS-Befehl gerichtet wird. Der STRING besteht
	aus sechs, durch Punkte getrennten Zahlenfeldern.
	Jedes Zahlenfeld enthäLT eine Zahl zwischen 0 und
	254. Gültige AMS-Netzwerkadressen sind z.B.
	"1.1.1.2.7.1" oder "200.5.7.170.1.7". Wird ein
	Leerstring übergeben, so wird automatisch die
	AMS-Netzwerkkennung des lokalen Gerätes angenommen.

*)
	sNetId 		: T_AmsNetId := '';
	bExecute 	: BOOL;
	nSlaveAddr 	: UINT := 1006;
	nIndex 		: WORD := 16#1018;
	nSubIndex 	: BYTE := 1;
	vendorId	: UDINT;
	bError 		: BOOL;
	nErrId 		: UDINT;
END_VAR
execTrigger(CLK := EXECUTE);
IF EXECUTE = FALSE THEN
	RETURN;
END_IF
IF execTrigger.Q = TRUE THEN   (* init *)
	busy := TRUE;
END_IF

fbSdoRead(sNetId := sNetId,
	nSlaveAddr := nSlaveAddr, nIndex := nIndex, nSubIndex := nSubIndex,
	pDstBuf := ADR(vendorId), cbBufLen := SIZEOF(vendorId),
	bExecute := bExecute);
bError := fbSdoRead.bError;
nErrId := fbSdoRead.nErrId;
END_FUNCTION_BLOCK

(* POU FBs/FB_Froeling, ST *)
FUNCTION_BLOCK FB_Froeling
(*
	baudrate setting: not supported by this FB yet
		seems to be fixed at 57600 baud on froeling
		manually configure this and the following on the terminal!
	8N1
	no handshake
	--> a 3-wire connection (RX, TX, GND) on froeling COM2 should be sufficient
	
	set the protocol on froeling to RTU! (ASCII is not supported by this code currently)

	all values are transmitted as 16bit signed integers
*)

(* register description
	00001..00031 Read Coil Status     (FC=01) 00001-00140
	10001..10003 Read Input Status    (FC=02) 10001-10075
	30001..30264 Read Input Registers (FC=04) 30001-30264
	33001..33020 Read Input Registers (FC=04) 33001-33020
	34001..34002 Read Input Registers (FC=04) 34001-34002
	40029..40493 Read Holding Registers (FC=03) 40001-40915
	
	Es können alle Parameter geschrieben werden (ab Software V50.04 B05.06).
	Write Single Register (FC=06) 40001-40915
*)
VAR_INPUT
	baudrate: UINT := 57600; (* unused yet - configure it manually on the terminal! *)
	modbusSlaveAddress: USINT; (* can be configured on froeling from 1 to 247 *)
	timeout: TIME := t#5s; (* TODO: default timeout should depend on the baudrate *)
END_VAR
VAR_OUTPUT
	modbusMasterBusy: BOOL;
	modbusMasterError: BOOL;
	modbusMasterErrorId: MODBUS_ERRORS;
	modbusMasterBytesRead: UINT;
	values: ARRAY [0..99] OF INT;
	Stoerung: BOOL;
	Heizkreis0_PumpeEin: BOOL;
	Heizkreis1_PumpeEin: BOOL;
	Heizkreis2_PumpeEin: BOOL;
	Heizkreis3_PumpeEin: BOOL;
	Heizkreis4_PumpeEin: BOOL;
	Heizkreis1_MischerAuf: BOOL;
	Heizkreis2_MischerAuf: BOOL;
	Heizkreis3_MischerAuf: BOOL;
	Heizkreis4_MischerAuf: BOOL;
	Heizkreis1_MischerZu: BOOL;
	Heizkreis2_MischerZu: BOOL;
	Heizkreis3_MischerZu: BOOL;
	Heizkreis4_MischerZu: BOOL;
	TuerOffen: BOOL;
	STB: BOOL;
	NotAus: BOOL;
	KesselTemperatur: REAL;
	AbgasTemperatur: REAL;
	BoardTemperatur: REAL;
	RestSauerstoff: REAL;
	AussenTemperatur: REAL;
	SaugzugDrehzahl: REAL;
	StbTemperatur: REAL;
	Fuehler2Temperatur: REAL;
	Saugzug: REAL;
	Kesselstellgroesse: REAL;
	Heizkreis1_VoraufIst: REAL;
	Heizkreis1_VoraufSoll: REAL;
	Heizkreis1_Party: UINT;
	Heizkreis1_RaumTemperatur: REAL;
	Heizkreis2_VoraufIst: REAL;
	Heizkreis2_VoraufSoll: REAL;
	Heizkreis2_Party: UINT;
	Heizkreis2_RaumTemperatur: REAL;
	Heizkreis3_VoraufIst: REAL;
	Heizkreis3_VoraufSoll: REAL;
	Heizkreis3_Party: UINT;
	Heizkreis3_RaumTemperatur: REAL;
	Heizkreis4_VoraufIst: REAL;
	Heizkreis4_VoraufSoll: REAL;
	Heizkreis4_Party: UINT;
	Heizkreis4_RaumTemperatur: REAL;

	Boiler1_TemperaturOben: REAL;
	Boiler1_TemperaturSolarreferenz: REAL;
	Board_TemperaturPelletmodul: REAL;
	Betriebsstunden: INT;
	Boiler2_ObenTemperatur: REAL;
	Boiler2_SolarreferenzTemperatur: REAL;
	Boiler3_ObenTemperatur: REAL;
	Boiler3_SolarreferenzTemperatur: REAL;
	Boiler4_ObenTemperatur: REAL;
	Boiler4_SolarreferenzTemperatur: REAL;
	Puffer1_ObenTemperatur: REAL;
	Puffer1_MitteTemperatur: REAL;
	Puffer1_UntenTemperatur: REAL;
	Puffer2_ObenTemperatur: REAL;
	Puffer2_MitteTemperatur: REAL;
	Puffer2_UntenTemperatur: REAL;
	Puffer3_ObenTemperatur: REAL;
	Puffer3_MitteTemperatur: REAL;
	Puffer3_UntenTemperatur: REAL;
	Puffer4_ObenTemperatur: REAL;
	Puffer4_MitteTemperatur: REAL;
	Puffer4_UntenTemperatur: REAL;
	Kessel_SollTemperatur: REAL;
	Solarfuehler_PufferuntenTemperatur: REAL;
	Puffer1_Pumpe: REAL;
	Puffer2_Pumpe: REAL;
	Puffer3_Pumpe: REAL;
	Puffer4_Pumpe: REAL;
	Boiler1_Pumpe: REAL;
	Boiler2_Pumpe: REAL;
	Boiler3_Pumpe: REAL;
	Boiler4_Pumpe: REAL;
	Kollektor_Pumpe: REAL;
	Abgas_Soll_Temperatur: REAL;
	Kollektor_Temperatur: REAL;
	Kollektor_Pumpe_Laufzeit: UINT;
	Kollektor_Ruecklauf_Temperatur: REAL;
	Kessel_Anforderung: BOOL;
	Heizen_Stunden: UINT;
	Solar_BoilerUnten_Temperatur: REAL;
	Solar_Leistung: REAL;

	Kessel_Soll_Temperatur: REAL;

	AnlagenZustand: E_FroelingAnlagenzustand;
	KesselZustand: E_FroelingKesselzustand;
END_VAR
VAR
	initOnce: BOOL := TRUE;
	initScan: BOOL := TRUE;
	modbusMaster: ModbusRtuMaster_KL6x22B;
	modbusMasterReadyTrigger: F_TRIG;
	i: UINT;
	j: UINT;
	offset: UINT;
	length: UINT;
	n: USINT;
	execute: BOOL;
	setValues: BOOL;
END_VAR

VAR CONSTANT
	addresses: ARRAY [0..7] OF ST_ModbusAddressRange :=
		(start := 0, length := 8, accessFunction := ReadCoils),
		(start := 8, length := 8, accessFunction := ReadCoils),
		(start := 16, length := 8, accessFunction := ReadCoils),
		(start := 24, length := 8, accessFunction := ReadCoils),
		(start := 0, length := 8, accessFunction := ReadInputStatus),
		(start := 0, length := 37, accessFunction := ReadInputRegs),
		(start := 93, length := 12, accessFunction := ReadInputRegs),
		(start := 4000, length := 3, accessFunction := ReadInputRegs);
	dummyAddress: ST_ModbusAddressRange;
END_VAR
IF initOnce THEN   (* TODO: howto detect an online change? *)
	n := SIZEOF(addresses) / SIZEOF(dummyAddress);
	modbusMaster.UnitID := modbusSlaveAddress;
	modbusMaster.Timeout := timeout;
	initOnce := FALSE;
END_IF

IF initScan THEN
	i := 0;
	offset := 0;
	execute := TRUE;
END_IF

